LIN {X -0.115,Y -453.231,Z 768.523,A 0.000,B 0.000,C 90.000,E1 94.188} C_DIS
LIN {X 0.209,Y -441.249,Z 768.512,A 0.000,B 0.000,C 90.000,E1 92.064} C_DIS
LIN {X -0.076,Y -432.103,Z 768.503,A 0.000,B 0.000,C 90.000,E1 90.516} C_DIS
LIN {X -0.093,Y -422.619,Z 768.494,A 0.000,B 0.000,C 90.000,E1 88.912} C_DIS
LIN {X -0.178,Y -411.419,Z 768.483,A 0.000,B 0.000,C 90.000,E1 87.020} C_DIS
LIN {X -0.031,Y -400.090,Z 768.473,A 0.000,B 0.000,C 90.000,E1 85.065} C_DIS
LIN {X -0.072,Y -387.195,Z 768.460,A 0.000,B 0.000,C 90.000,E1 82.818} C_DIS
LIN {X 0.067,Y -373.104,Z 768.446,A 0.000,B 0.000,C 90.000,E1 80.208} C_DIS
LIN {X -0.105,Y -356.698,Z 768.428,A 0.000,B 0.000,C 90.000,E1 76.992} C_DIS
LIN {X -0.066,Y -345.249,Z 768.414,A 0.000,B 0.000,C 90.000,E1 74.574} C_DIS
LIN {X -0.147,Y -332.594,Z 768.399,A 0.000,B 0.000,C 90.000,E1 71.819} C_DIS
LIN {X 0.059,Y -320.333,Z 768.383,A 0.000,B 0.000,C 90.000,E1 68.954} C_DIS
LIN {X 0.088,Y -306.265,Z 768.363,A 0.000,B 0.000,C 90.000,E1 65.409} C_DIS
LIN {X 0.158,Y -293.532,Z 768.343,A 0.000,B 0.000,C 90.000,E1 61.769} C_DIS
LIN {X -0.092,Y -282.992,Z 768.325,A 0.000,B 0.000,C 90.000,E1 58.456} C_DIS
LIN {X 0.131,Y -275.046,Z 768.309,A 0.000,B 0.000,C 90.000,E1 55.674} C_DIS
LIN {X 0.000,Y -269.175,Z 768.298,A 0.000,B 0.000,C 90.000,E1 53.623} C_DIS
LIN {X 0.052,Y -261.369,Z 768.282,A 0.000,B 0.000,C 90.000,E1 50.803} C_DIS
LIN {X -0.041,Y -255.557,Z 768.270,A 0.000,B 0.000,C 90.000,E1 48.690} C_DIS
LIN {X -0.056,Y -247.855,Z 768.254,A 0.000,B 0.000,C 90.000,E1 45.810} C_DIS
LIN {X 0.075,Y -240.330,Z 768.238,A 0.000,B 0.000,C 90.000,E1 42.852} C_DIS
LIN {X 0.127,Y -231.043,Z 768.217,A 0.000,B 0.000,C 90.000,E1 39.116} C_DIS
LIN {X -0.014,Y -222.274,Z 768.196,A 0.000,B 0.000,C 90.000,E1 35.358} C_DIS
LIN {X 0.103,Y -214.211,Z 768.175,A 0.000,B 0.000,C 90.000,E1 31.465} C_DIS
LIN {X -0.013,Y -208.482,Z 768.158,A 0.000,B 0.000,C 90.000,E1 28.359} C_DIS
LIN {X 0.089,Y -203.532,Z 768.140,A 0.000,B 0.000,C 90.000,E1 25.155} C_DIS
LIN {X 0.040,Y -198.253,Z 768.118,A 0.000,B 0.000,C 90.000,E1 21.153} C_DIS
LIN {X 0.031,Y -194.129,Z 768.095,A 0.000,B 0.000,C 90.000,E1 17.094} C_DIS
LIN {X -0.008,Y -190.564,Z 768.068,A 0.000,B 0.000,C 90.000,E1 12.187} C_DIS
LIN {X 0.018,Y -188.134,Z 768.031,A 0.000,B 0.000,C 90.000,E1 5.568} C_DIS
LIN {X 0.043,Y -189.539,Z 767.970,A 0.000,B 0.000,C 90.000,E1 354.546} C_DIS
LIN {X -0.098,Y -193.008,Z 767.938,A 0.000,B 0.000,C 90.000,E1 348.814} C_DIS
LIN {X -0.033,Y -196.683,Z 767.915,A 0.000,B 0.000,C 90.000,E1 344.700} C_DIS
LIN {X 0.094,Y -201.414,Z 767.892,A 0.000,B 0.000,C 90.000,E1 340.604} C_DIS
LIN {X 0.009,Y -207.080,Z 767.870,A 0.000,B 0.000,C 90.000,E1 336.613} C_DIS
LIN {X -0.054,Y -213.642,Z 767.848,A 0.000,B 0.000,C 90.000,E1 332.666} C_DIS
LIN {X 0.008,Y -221.031,Z 767.826,A 0.000,B 0.000,C 90.000,E1 328.742} C_DIS
LIN {X 0.008,Y -228.997,Z 767.805,A 0.000,B 0.000,C 90.000,E1 324.895} C_DIS
LIN {X 0.108,Y -237.690,Z 767.784,A 0.000,B 0.000,C 90.000,E1 321.090} C_DIS
LIN {X 0.044,Y -247.109,Z 767.763,A 0.000,B 0.000,C 90.000,E1 317.391} C_DIS
LIN {X -0.092,Y -257.488,Z 767.743,A 0.000,B 0.000,C 90.000,E1 313.785} C_DIS
LIN {X 0.081,Y -267.584,Z 767.725,A 0.000,B 0.000,C 90.000,E1 310.539} C_DIS
LIN {X -0.049,Y -279.903,Z 767.706,A 0.000,B 0.000,C 90.000,E1 307.076} C_DIS
LIN {X 0.000,Y -293.440,Z 767.687,A 0.000,B 0.000,C 90.000,E1 303.658} C_DIS
LIN {X -0.087,Y -302.469,Z 767.676,A 0.000,B 0.000,C 90.000,E1 301.671} C_DIS
LIN {X 0.173,Y -319.454,Z 767.658,A 0.000,B 0.000,C 90.000,E1 298.359} C_DIS
LIN {X 0.007,Y -334.044,Z 767.644,A 0.000,B 0.000,C 90.000,E1 295.848} C_DIS
LIN {X 0.203,Y -345.763,Z 767.633,A 0.000,B 0.000,C 90.000,E1 293.951} C_DIS
LIN {X -0.078,Y -366.819,Z 767.616,A 0.000,B 0.000,C 90.000,E1 290.972} C_DIS
LIN {X -0.107,Y -390.144,Z 767.600,A 0.000,B 0.000,C 90.000,E1 288.055} C_DIS
LIN {X -0.085,Y -407.451,Z 767.589,A 0.000,B 0.000,C 90.000,E1 286.079} C_DIS
LIN {X 0.167,Y -419.629,Z 767.582,A 0.000,B 0.000,C 90.000,E1 284.662} C_DIS
LIN {X 0.199,Y -431.468,Z 767.574,A 0.000,B 0.000,C 90.000,E1 283.300} C_DIS
LIN {X -0.116,Y -442.966,Z 767.567,A 0.000,B 0.000,C 90.000,E1 282.007} C_DIS
LIN {X -0.085,Y -451.698,Z 767.561,A 0.000,B 0.000,C 90.000,E1 280.950} C_DIS
LIN {X 0.236,Y -461.835,Z 767.554,A 0.000,B 0.000,C 90.000,E1 279.613} C_DIS
LIN {X -0.050,Y -469.557,Z 767.548,A 0.000,B 0.000,C 90.000,E1 278.624} C_DIS
LIN {X -0.112,Y -475.010,Z 767.544,A 0.000,B 0.000,C 90.000,E1 277.871} C_DIS
LIN {X -0.194,Y -479.966,Z 767.539,A 0.000,B 0.000,C 90.000,E1 277.125} C_DIS
LIN {X -0.166,Y -484.180,Z 767.535,A 0.000,B 0.000,C 90.000,E1 276.372} C_DIS
LIN {X 0.012,Y -486.561,Z 767.533,A 0.000,B 0.000,C 90.000,E1 275.853} C_DIS
LIN {X 0.043,Y -489.431,Z 767.528,A 0.000,B 0.000,C 90.000,E1 275.106} C_DIS
LIN {X 0.251,Y -490.885,Z 767.526,A 0.000,B 0.000,C 90.000,E1 274.588} C_DIS
LIN {X -0.058,Y -491.996,Z 767.523,A 0.000,B 0.000,C 90.000,E1 274.131} C_DIS
LIN {X 0.168,Y -492.709,Z 767.520,A 0.000,B 0.000,C 90.000,E1 273.612} C_DIS
LIN {X -0.122,Y -493.040,Z 767.517,A 0.000,B 0.000,C 90.000,E1 273.154} C_DIS
LIN {X 0.111,Y -492.940,Z 767.515,A 0.000,B 0.000,C 90.000,E1 272.636} C_DIS
LIN {X -0.171,Y -492.377,Z 767.512,A 0.000,B 0.000,C 90.000,E1 272.178} C_DIS
LIN {X 0.057,Y -491.366,Z 767.509,A 0.000,B 0.000,C 90.000,E1 271.661} C_DIS
LIN {X -0.226,Y -489.879,Z 767.507,A 0.000,B 0.000,C 90.000,E1 271.203} C_DIS
LIN {X -0.023,Y -487.905,Z 767.504,A 0.000,B 0.000,C 90.000,E1 270.688} C_DIS
LIN {X 0.170,Y -485.305,Z 767.501,A 0.000,B 0.000,C 90.000,E1 270.172} C_DIS
LIN {X -0.139,Y -482.169,Z 767.498,A 0.000,B 0.000,C 90.000,E1 269.714} C_DIS
LIN {X 0.018,Y -478.202,Z 767.496,A 0.000,B 0.000,C 90.000,E1 269.198} C_DIS
LIN {X 0.152,Y -473.377,Z 767.493,A 0.000,B 0.000,C 90.000,E1 268.682} C_DIS
LIN {X -0.152,Y -467.577,Z 767.490,A 0.000,B 0.000,C 90.000,E1 268.224} C_DIS
LIN {X 0.054,Y -461.202,Z 767.488,A 0.000,B 0.000,C 90.000,E1 267.764} C_DIS
LIN {X -0.042,Y -457.997,Z 767.487,A 0.000,B 0.000,C 90.000,E1 267.593} C_DIS
LIN {X -0.137,Y -454.304,Z 767.486,A 0.000,B 0.000,C 90.000,E1 267.421} C_DIS
LIN {X -0.211,Y -446.988,Z 767.484,A 0.000,B 0.000,C 90.000,E1 267.135} C_DIS
LIN {X 0.167,Y -438.672,Z 767.483,A 0.000,B 0.000,C 90.000,E1 266.849} C_DIS
LIN {X -0.167,Y -429.640,Z 767.482,A 0.000,B 0.000,C 90.000,E1 266.731} C_DIS
LIN {X 0.129,Y -422.215,Z 767.481,A 0.000,B 0.000,C 90.000,E1 266.617} C_DIS
LIN {X 0.019,Y -417.823,Z 767.481,A 0.000,B 0.000,C 90.000,E1 266.617} C_DIS
LIN {X -0.015,Y -180.956,Z 767.481,A 0.000,B 0.000,C 90.000,E1 266.617} C_DIS
LIN {X 0.065,Y -180.879,Z 767.473,A 0.000,B 0.000,C 90.000,E1 265.065} C_DIS
LIN {X 0.006,Y -178.802,Z 767.442,A 0.000,B 0.000,C 90.000,E1 259.511} C_DIS
LIN {X 0.082,Y -175.847,Z 767.413,A 0.000,B 0.000,C 90.000,E1 254.393} C_DIS
LIN {X 0.042,Y -172.583,Z 767.390,A 0.000,B 0.000,C 90.000,E1 250.134} C_DIS
LIN {X 0.058,Y -171.470,Z 767.380,A 0.000,B 0.000,C 90.000,E1 248.411} C_DIS
LIN {X 0.038,Y -167.702,Z 767.356,A 0.000,B 0.000,C 90.000,E1 244.101} C_DIS
LIN {X 0.051,Y -166.387,Z 767.347,A 0.000,B 0.000,C 90.000,E1 242.359} C_DIS
LIN {X 0.042,Y -163.114,Z 767.327,A 0.000,B 0.000,C 90.000,E1 238.869} C_DIS
LIN {X 0.093,Y -161.064,Z 767.313,A 0.000,B 0.000,C 90.000,E1 236.215} C_DIS
LIN {X -0.021,Y -157.798,Z 767.293,A 0.000,B 0.000,C 90.000,E1 232.718} C_DIS
LIN {X 0.019,Y -155.834,Z 767.278,A 0.000,B 0.000,C 90.000,E1 230.033} C_DIS
LIN {X -0.024,Y -152.084,Z 767.253,A 0.000,B 0.000,C 90.000,E1 225.567} C_DIS
LIN {X -0.006,Y -150.334,Z 767.238,A 0.000,B 0.000,C 90.000,E1 222.852} C_DIS
LIN {X 0.015,Y -147.074,Z 767.213,A 0.000,B 0.000,C 90.000,E1 218.302} C_DIS
LIN {X -0.081,Y -145.648,Z 767.198,A 0.000,B 0.000,C 90.000,E1 215.598} C_DIS
LIN {X -0.077,Y -143.031,Z 767.172,A 0.000,B 0.000,C 90.000,E1 211.003} C_DIS
LIN {X 0.050,Y -141.656,Z 767.152,A 0.000,B 0.000,C 90.000,E1 207.257} C_DIS
LIN {X -0.031,Y -139.445,Z 767.115,A 0.000,B 0.000,C 90.000,E1 200.791} C_DIS
LIN {X 0.022,Y -139.179,Z 767.105,A 0.000,B 0.000,C 90.000,E1 198.906} C_DIS
LIN {X 0.050,Y -138.320,Z 767.053,A 0.000,B 0.000,C 90.000,E1 189.557} C_DIS
LIN {X 0.059,Y -139.466,Z 767.007,A 0.000,B 0.000,C 90.000,E1 181.146} C_DIS
LIN {X 0.001,Y -141.031,Z 766.975,A 0.000,B 0.000,C 90.000,E1 175.584} C_DIS
LIN {X -0.046,Y -142.398,Z 766.960,A 0.000,B 0.000,C 90.000,E1 172.818} C_DIS
LIN {X 0.017,Y -144.630,Z 766.934,A 0.000,B 0.000,C 90.000,E1 168.173} C_DIS
LIN {X 0.077,Y -147.825,Z 766.909,A 0.000,B 0.000,C 90.000,E1 163.559} C_DIS
LIN {X 0.022,Y -150.517,Z 766.889,A 0.000,B 0.000,C 90.000,E1 159.934} C_DIS
LIN {X 0.043,Y -153.979,Z 766.868,A 0.000,B 0.000,C 90.000,E1 156.305} C_DIS
LIN {X -0.037,Y -157.391,Z 766.849,A 0.000,B 0.000,C 90.000,E1 152.743} C_DIS
LIN {X 0.043,Y -161.596,Z 766.829,A 0.000,B 0.000,C 90.000,E1 149.154} C_DIS
LIN {X -0.085,Y -165.793,Z 766.809,A 0.000,B 0.000,C 90.000,E1 145.674} C_DIS
LIN {X 0.035,Y -170.756,Z 766.790,A 0.000,B 0.000,C 90.000,E1 142.145} C_DIS
LIN {X 0.058,Y -175.628,Z 766.771,A 0.000,B 0.000,C 90.000,E1 138.690} C_DIS
LIN {X -0.073,Y -181.243,Z 766.752,A 0.000,B 0.000,C 90.000,E1 135.324} C_DIS
LIN {X 0.058,Y -186.714,Z 766.733,A 0.000,B 0.000,C 90.000,E1 131.919} C_DIS
LIN {X 0.072,Y -191.544,Z 766.718,A 0.000,B 0.000,C 90.000,E1 129.277} C_DIS
LIN {X 0.081,Y -192.281,Z 766.716,A 0.000,B 0.000,C 90.000,E1 128.830} C_DIS
LIN {X 0.083,Y -291.983,Z 766.716,A 0.000,B 0.000,C 90.000,E1 128.830} C_DIS
LIN {X -0.037,Y -293.381,Z 766.716,A 0.000,B 0.000,C 90.000,E1 128.830} C_DIS
LIN {X -0.045,Y -297.878,Z 766.715,A 0.000,B 0.000,C 90.000,E1 128.624} C_DIS
LIN {X -0.048,Y -301.099,Z 766.713,A 0.000,B 0.000,C 90.000,E1 128.338} C_DIS
LIN {X 0.011,Y -304.766,Z 766.710,A 0.000,B 0.000,C 90.000,E1 127.810} C_DIS
LIN {X -0.036,Y -306.408,Z 766.708,A 0.000,B 0.000,C 90.000,E1 127.488} C_DIS
LIN {X -0.027,Y -307.697,Z 766.706,A 0.000,B 0.000,C 90.000,E1 127.156} C_DIS
LIN {X 0.075,Y -319.692,Z 766.685,A 0.000,B 0.000,C 90.000,E1 123.245} C_DIS
LIN {X 0.074,Y -330.066,Z 766.669,A 0.000,B 0.000,C 90.000,E1 120.384} C_DIS
LIN {X -0.017,Y -341.793,Z 766.653,A 0.000,B 0.000,C 90.000,E1 117.590} C_DIS
LIN {X 0.075,Y -354.971,Z 766.638,A 0.000,B 0.000,C 90.000,E1 114.823} C_DIS
LIN {X -0.138,Y -368.003,Z 766.625,A 0.000,B 0.000,C 90.000,E1 112.461} C_DIS
LIN {X -0.165,Y -382.370,Z 766.612,A 0.000,B 0.000,C 90.000,E1 110.120} C_DIS
LIN {X -0.096,Y -398.176,Z 766.599,A 0.000,B 0.000,C 90.000,E1 107.819} C_DIS
LIN {X 0.141,Y -415.535,Z 766.586,A 0.000,B 0.000,C 90.000,E1 105.552} C_DIS
LIN {X -0.101,Y -434.557,Z 766.574,A 0.000,B 0.000,C 90.000,E1 103.411} C_DIS
LIN {X -0.078,Y -454.655,Z 766.563,A 0.000,B 0.000,C 90.000,E1 101.366} C_DIS
LIN {X 0.205,Y -467.509,Z 766.556,A 0.000,B 0.000,C 90.000,E1 100.141} C_DIS
LIN {X -0.231,Y -469.681,Z 766.555,A 0.000,B 0.000,C 90.000,E1 99.962} C_DIS
LIN {X -0.207,Y -471.323,Z 766.554,A 0.000,B 0.000,C 90.000,E1 99.726} C_DIS
LIN {X 0.033,Y -472.685,Z 766.552,A 0.000,B 0.000,C 90.000,E1 99.443} C_DIS
LIN {X -0.113,Y -473.694,Z 766.551,A 0.000,B 0.000,C 90.000,E1 99.208} C_DIS
LIN {X 0.074,Y -474.848,Z 766.548,A 0.000,B 0.000,C 90.000,E1 98.681} C_DIS
LIN {X 0.194,Y -475.004,Z 766.545,A 0.000,B 0.000,C 90.000,E1 98.163} C_DIS
LIN {X -0.147,Y -474.191,Z 766.543,A 0.000,B 0.000,C 90.000,E1 97.701} C_DIS
LIN {X -0.015,Y -472.276,Z 766.540,A 0.000,B 0.000,C 90.000,E1 97.182} C_DIS
LIN {X 0.113,Y -469.117,Z 766.537,A 0.000,B 0.000,C 90.000,E1 96.663} C_DIS
LIN {X 0.197,Y -451.453,Z 766.521,A 0.000,B 0.000,C 90.000,E1 93.841} C_DIS
LIN {X -0.173,Y -441.001,Z 766.511,A 0.000,B 0.000,C 90.000,E1 92.064} C_DIS
LIN {X -0.022,Y -431.870,Z 766.503,A 0.000,B 0.000,C 90.000,E1 90.458} C_DIS
LIN {X -0.044,Y -422.368,Z 766.494,A 0.000,B 0.000,C 90.000,E1 88.854} C_DIS
LIN {X -0.137,Y -411.187,Z 766.483,A 0.000,B 0.000,C 90.000,E1 86.963} C_DIS
LIN {X 0.004,Y -399.867,Z 766.472,A 0.000,B 0.000,C 90.000,E1 85.008} C_DIS
LIN {X -0.045,Y -386.980,Z 766.460,A 0.000,B 0.000,C 90.000,E1 82.761} C_DIS
LIN {X 0.092,Y -371.356,Z 766.444,A 0.000,B 0.000,C 90.000,E1 79.859} C_DIS
LIN {X -0.098,Y -356.521,Z 766.427,A 0.000,B 0.000,C 90.000,E1 76.937} C_DIS
LIN {X -0.067,Y -345.091,Z 766.414,A 0.000,B 0.000,C 90.000,E1 74.519} C_DIS
LIN {X -0.157,Y -332.443,Z 766.399,A 0.000,B 0.000,C 90.000,E1 71.764} C_DIS
LIN {X 0.040,Y -320.223,Z 766.383,A 0.000,B 0.000,C 90.000,E1 68.901} C_DIS
LIN {X 0.059,Y -306.215,Z 766.363,A 0.000,B 0.000,C 90.000,E1 65.357} C_DIS
LIN {X -0.137,Y -293.572,Z 766.343,A 0.000,B 0.000,C 90.000,E1 61.769} C_DIS
LIN {X -0.134,Y -283.092,Z 766.324,A 0.000,B 0.000,C 90.000,E1 58.408} C_DIS
LIN {X -0.140,Y -275.193,Z 766.309,A 0.000,B 0.000,C 90.000,E1 55.674} C_DIS
LIN {X 0.118,Y -267.422,Z 766.294,A 0.000,B 0.000,C 90.000,E1 52.844} C_DIS
LIN {X 0.169,Y -261.602,Z 766.282,A 0.000,B 0.000,C 90.000,E1 50.723} C_DIS
LIN {X 0.077,Y -255.815,Z 766.270,A 0.000,B 0.000,C 90.000,E1 48.609} C_DIS
LIN {X 0.066,Y -248.116,Z 766.254,A 0.000,B 0.000,C 90.000,E1 45.729} C_DIS
LIN {X 0.025,Y -240.586,Z 766.238,A 0.000,B 0.000,C 90.000,E1 42.813} C_DIS
LIN {X -0.006,Y -233.076,Z 766.221,A 0.000,B 0.000,C 90.000,E1 39.850} C_DIS
LIN {X 0.031,Y -225.925,Z 766.205,A 0.000,B 0.000,C 90.000,E1 36.824} C_DIS
LIN {X -0.032,Y -217.524,Z 766.183,A 0.000,B 0.000,C 90.000,E1 33.007} C_DIS
LIN {X 0.039,Y -211.441,Z 766.166,A 0.000,B 0.000,C 90.000,E1 29.873} C_DIS
LIN {X -0.058,Y -206.090,Z 766.148,A 0.000,B 0.000,C 90.000,E1 26.744} C_DIS
LIN {X 0.060,Y -200.405,Z 766.126,A 0.000,B 0.000,C 90.000,E1 22.717} C_DIS
LIN {X 0.072,Y -195.833,Z 766.104,A 0.000,B 0.000,C 90.000,E1 18.671} C_DIS
LIN {X 0.060,Y -192.317,Z 766.081,A 0.000,B 0.000,C 90.000,E1 14.592} C_DIS
LIN {X -0.041,Y -189.168,Z 766.049,A 0.000,B 0.000,C 90.000,E1 8.859} C_DIS
LIN {X -0.028,Y -190.058,Z 765.965,A 0.000,B 0.000,C 90.000,E1 353.742} C_DIS
LIN {X -0.087,Y -193.131,Z 765.938,A 0.000,B 0.000,C 90.000,E1 348.814} C_DIS
LIN {X -0.018,Y -196.809,Z 765.915,A 0.000,B 0.000,C 90.000,E1 344.700} C_DIS
LIN {X 0.113,Y -201.538,Z 765.892,A 0.000,B 0.000,C 90.000,E1 340.604} C_DIS
LIN {X 0.032,Y -207.205,Z 765.870,A 0.000,B 0.000,C 90.000,E1 336.613} C_DIS
LIN {X -0.027,Y -213.763,Z 765.848,A 0.000,B 0.000,C 90.000,E1 332.666} C_DIS
LIN {X 0.040,Y -221.120,Z 765.826,A 0.000,B 0.000,C 90.000,E1 328.742} C_DIS
LIN {X 0.045,Y -229.078,Z 765.805,A 0.000,B 0.000,C 90.000,E1 324.895} C_DIS
LIN {X -0.001,Y -237.750,Z 765.784,A 0.000,B 0.000,C 90.000,E1 321.126} C_DIS
LIN {X 0.089,Y -247.144,Z 765.763,A 0.000,B 0.000,C 90.000,E1 317.391} C_DIS
LIN {X -0.044,Y -257.529,Z 765.743,A 0.000,B 0.000,C 90.000,E1 313.785} C_DIS
LIN {X 0.131,Y -267.596,Z 765.725,A 0.000,B 0.000,C 90.000,E1 310.539} C_DIS
LIN {X 0.004,Y -279.903,Z 765.706,A 0.000,B 0.000,C 90.000,E1 307.076} C_DIS
LIN {X 0.056,Y -293.422,Z 765.687,A 0.000,B 0.000,C 90.000,E1 303.658} C_DIS
LIN {X -0.031,Y -302.437,Z 765.676,A 0.000,B 0.000,C 90.000,E1 301.671} C_DIS
LIN {X -0.050,Y -319.412,Z 765.658,A 0.000,B 0.000,C 90.000,E1 298.409} C_DIS
LIN {X 0.032,Y -335.868,Z 765.642,A 0.000,B 0.000,C 90.000,E1 295.540} C_DIS
LIN {X 0.045,Y -355.974,Z 765.625,A 0.000,B 0.000,C 90.000,E1 292.461} C_DIS
LIN {X -0.157,Y -375.747,Z 765.610,A 0.000,B 0.000,C 90.000,E1 289.812} C_DIS
LIN {X 0.051,Y -399.750,Z 765.594,A 0.000,B 0.000,C 90.000,E1 286.913} C_DIS
LIN {X -0.113,Y -412.105,Z 765.586,A 0.000,B 0.000,C 90.000,E1 285.536} C_DIS
LIN {X 0.208,Y -424.131,Z 765.579,A 0.000,B 0.000,C 90.000,E1 284.120} C_DIS
LIN {X -0.221,Y -435.815,Z 765.571,A 0.000,B 0.000,C 90.000,E1 282.827} C_DIS
LIN {X 0.160,Y -444.933,Z 765.565,A 0.000,B 0.000,C 90.000,E1 281.715} C_DIS
LIN {X 0.219,Y -453.492,Z 765.559,A 0.000,B 0.000,C 90.000,E1 280.658} C_DIS
LIN {X 0.124,Y -463.520,Z 765.552,A 0.000,B 0.000,C 90.000,E1 279.378} C_DIS
LIN {X -0.219,Y -471.181,Z 765.547,A 0.000,B 0.000,C 90.000,E1 278.398} C_DIS
LIN {X 0.202,Y -476.526,Z 765.542,A 0.000,B 0.000,C 90.000,E1 277.587} C_DIS
LIN {X 0.204,Y -481.299,Z 765.538,A 0.000,B 0.000,C 90.000,E1 276.834} C_DIS
LIN {X 0.186,Y -485.273,Z 765.534,A 0.000,B 0.000,C 90.000,E1 276.087} C_DIS
LIN {X -0.108,Y -487.531,Z 765.531,A 0.000,B 0.000,C 90.000,E1 275.625} C_DIS
LIN {X 0.094,Y -489.377,Z 765.528,A 0.000,B 0.000,C 90.000,E1 275.106} C_DIS
LIN {X -0.187,Y -490.862,Z 765.526,A 0.000,B 0.000,C 90.000,E1 274.645} C_DIS
LIN {X -0.006,Y -492.002,Z 765.523,A 0.000,B 0.000,C 90.000,E1 274.131} C_DIS
LIN {X 0.219,Y -492.762,Z 765.520,A 0.000,B 0.000,C 90.000,E1 273.612} C_DIS
LIN {X -0.071,Y -493.127,Z 765.517,A 0.000,B 0.000,C 90.000,E1 273.154} C_DIS
LIN {X 0.162,Y -493.046,Z 765.515,A 0.000,B 0.000,C 90.000,E1 272.636} C_DIS
LIN {X -0.119,Y -492.562,Z 765.512,A 0.000,B 0.000,C 90.000,E1 272.178} C_DIS
LIN {X 0.109,Y -491.565,Z 765.509,A 0.000,B 0.000,C 90.000,E1 271.661} C_DIS
LIN {X -0.173,Y -490.119,Z 765.507,A 0.000,B 0.000,C 90.000,E1 271.203} C_DIS
LIN {X 0.031,Y -488.140,Z 765.504,A 0.000,B 0.000,C 90.000,E1 270.688} C_DIS
LIN {X 0.225,Y -485.587,Z 765.501,A 0.000,B 0.000,C 90.000,E1 270.172} C_DIS
LIN {X -0.083,Y -482.401,Z 765.498,A 0.000,B 0.000,C 90.000,E1 269.714} C_DIS
LIN {X 0.076,Y -478.460,Z 765.496,A 0.000,B 0.000,C 90.000,E1 269.198} C_DIS
LIN {X 0.211,Y -473.627,Z 765.493,A 0.000,B 0.000,C 90.000,E1 268.682} C_DIS
LIN {X 0.081,Y -470.963,Z 765.491,A 0.000,B 0.000,C 90.000,E1 268.453} C_DIS
LIN {X 0.062,Y -465.020,Z 765.489,A 0.000,B 0.000,C 90.000,E1 267.993} C_DIS
LIN {X 0.046,Y -458.501,Z 765.487,A 0.000,B 0.000,C 90.000,E1 267.593} C_DIS
LIN {X 0.125,Y -451.362,Z 765.485,A 0.000,B 0.000,C 90.000,E1 267.249} C_DIS
LIN {X -0.140,Y -447.619,Z 765.484,A 0.000,B 0.000,C 90.000,E1 267.135} C_DIS
LIN {X 0.199,Y -439.329,Z 765.483,A 0.000,B 0.000,C 90.000,E1 266.849} C_DIS
LIN {X -0.167,Y -430.566,Z 765.482,A 0.000,B 0.000,C 90.000,E1 266.731} C_DIS
LIN {X 0.112,Y -423.768,Z 765.481,A 0.000,B 0.000,C 90.000,E1 266.617} C_DIS
LIN {X -0.065,Y -419.400,Z 765.481,A 0.000,B 0.000,C 90.000,E1 266.617} C_DIS
LIN {X -0.053,Y -180.956,Z 765.481,A 0.000,B 0.000,C 90.000,E1 266.617} C_DIS
LIN {X 0.026,Y -180.877,Z 765.473,A 0.000,B 0.000,C 90.000,E1 265.065} C_DIS
LIN {X -0.032,Y -178.795,Z 765.442,A 0.000,B 0.000,C 90.000,E1 259.511} C_DIS
LIN {X 0.044,Y -175.840,Z 765.413,A 0.000,B 0.000,C 90.000,E1 254.393} C_DIS
LIN {X 0.044,Y -172.032,Z 765.385,A 0.000,B 0.000,C 90.000,E1 249.263} C_DIS
LIN {X 0.020,Y -171.460,Z 765.380,A 0.000,B 0.000,C 90.000,E1 248.411} C_DIS
LIN {X 0.000,Y -167.692,Z 765.356,A 0.000,B 0.000,C 90.000,E1 244.101} C_DIS
LIN {X 0.014,Y -166.375,Z 765.346,A 0.000,B 0.000,C 90.000,E1 242.359} C_DIS
LIN {X 0.005,Y -163.104,Z 765.327,A 0.000,B 0.000,C 90.000,E1 238.869} C_DIS
LIN {X 0.056,Y -161.051,Z 765.312,A 0.000,B 0.000,C 90.000,E1 236.215} C_DIS
LIN {X 0.039,Y -157.787,Z 765.293,A 0.000,B 0.000,C 90.000,E1 232.683} C_DIS
LIN {X -0.017,Y -155.823,Z 765.278,A 0.000,B 0.000,C 90.000,E1 230.033} C_DIS
LIN {X -0.060,Y -152.074,Z 765.253,A 0.000,B 0.000,C 90.000,E1 225.567} C_DIS
LIN {X -0.041,Y -150.325,Z 765.238,A 0.000,B 0.000,C 90.000,E1 222.852} C_DIS
LIN {X -0.020,Y -147.066,Z 765.213,A 0.000,B 0.000,C 90.000,E1 218.302} C_DIS
LIN {X 0.088,Y -145.642,Z 765.198,A 0.000,B 0.000,C 90.000,E1 215.518} C_DIS
LIN {X 0.086,Y -143.025,Z 765.172,A 0.000,B 0.000,C 90.000,E1 210.924} C_DIS
LIN {X 0.017,Y -141.650,Z 765.151,A 0.000,B 0.000,C 90.000,E1 207.257} C_DIS
LIN {X -0.063,Y -139.444,Z 765.115,A 0.000,B 0.000,C 90.000,E1 200.791} C_DIS
LIN {X -0.011,Y -139.177,Z 765.105,A 0.000,B 0.000,C 90.000,E1 198.906} C_DIS
LIN {X 0.017,Y -138.319,Z 765.053,A 0.000,B 0.000,C 90.000,E1 189.557} C_DIS
LIN {X 0.026,Y -139.468,Z 765.006,A 0.000,B 0.000,C 90.000,E1 181.146} C_DIS
LIN {X -0.033,Y -141.036,Z 764.975,A 0.000,B 0.000,C 90.000,E1 175.584} C_DIS
LIN {X 0.062,Y -142.404,Z 764.960,A 0.000,B 0.000,C 90.000,E1 172.761} C_DIS
LIN {X -0.017,Y -144.638,Z 764.934,A 0.000,B 0.000,C 90.000,E1 168.173} C_DIS
LIN {X 0.043,Y -147.834,Z 764.909,A 0.000,B 0.000,C 90.000,E1 163.559} C_DIS
LIN {X -0.013,Y -150.529,Z 764.888,A 0.000,B 0.000,C 90.000,E1 159.934} C_DIS
LIN {X 0.007,Y -153.992,Z 764.868,A 0.000,B 0.000,C 90.000,E1 156.305} C_DIS
LIN {X -0.073,Y -157.406,Z 764.848,A 0.000,B 0.000,C 90.000,E1 152.743} C_DIS
LIN {X 0.007,Y -161.613,Z 764.829,A 0.000,B 0.000,C 90.000,E1 149.154} C_DIS
LIN {X 0.108,Y -165.809,Z 764.809,A 0.000,B 0.000,C 90.000,E1 145.595} C_DIS
LIN {X -0.003,Y -170.775,Z 764.790,A 0.000,B 0.000,C 90.000,E1 142.145} C_DIS
LIN {X 0.020,Y -175.647,Z 764.771,A 0.000,B 0.000,C 90.000,E1 138.690} C_DIS
LIN {X 0.018,Y -181.261,Z 764.752,A 0.000,B 0.000,C 90.000,E1 135.283} C_DIS
LIN {X 0.017,Y -186.735,Z 764.733,A 0.000,B 0.000,C 90.000,E1 131.919} C_DIS
LIN {X 0.032,Y -191.563,Z 764.718,A 0.000,B 0.000,C 90.000,E1 129.277} C_DIS
LIN {X -0.105,Y -192.238,Z 764.716,A 0.000,B 0.000,C 90.000,E1 128.910} C_DIS
LIN {X -0.022,Y -291.703,Z 764.716,A 0.000,B 0.000,C 90.000,E1 128.874} C_DIS
LIN {X 0.068,Y -293.365,Z 764.716,A 0.000,B 0.000,C 90.000,E1 128.830} C_DIS
LIN {X -0.108,Y -298.260,Z 764.714,A 0.000,B 0.000,C 90.000,E1 128.624} C_DIS
LIN {X -0.013,Y -301.459,Z 764.713,A 0.000,B 0.000,C 90.000,E1 128.302} C_DIS
LIN {X 0.139,Y -305.106,Z 764.710,A 0.000,B 0.000,C 90.000,E1 127.729} C_DIS
LIN {X -0.094,Y -306.656,Z 764.708,A 0.000,B 0.000,C 90.000,E1 127.443} C_DIS
LIN {X 0.103,Y -307.876,Z 764.706,A 0.000,B 0.000,C 90.000,E1 127.076} C_DIS
LIN {X 0.141,Y -318.779,Z 764.686,A 0.000,B 0.000,C 90.000,E1 123.499} C_DIS
LIN {X -0.062,Y -329.035,Z 764.670,A 0.000,B 0.000,C 90.000,E1 120.669} C_DIS
LIN {X -0.015,Y -340.630,Z 764.655,A 0.000,B 0.000,C 90.000,E1 117.847} C_DIS
LIN {X 0.040,Y -353.673,Z 764.639,A 0.000,B 0.000,C 90.000,E1 115.079} C_DIS
LIN {X -0.062,Y -366.572,Z 764.626,A 0.000,B 0.000,C 90.000,E1 112.695} C_DIS
LIN {X -0.132,Y -380.797,Z 764.613,A 0.000,B 0.000,C 90.000,E1 110.355} C_DIS
LIN {X -0.107,Y -396.448,Z 764.600,A 0.000,B 0.000,C 90.000,E1 108.055} C_DIS
LIN {X 0.079,Y -413.641,Z 764.588,A 0.000,B 0.000,C 90.000,E1 105.788} C_DIS
LIN {X 0.196,Y -432.500,Z 764.576,A 0.000,B 0.000,C 90.000,E1 103.592} C_DIS
LIN {X 0.182,Y -452.537,Z 764.564,A 0.000,B 0.000,C 90.000,E1 101.535} C_DIS
LIN {X -0.123,Y -467.906,Z 764.556,A 0.000,B 0.000,C 90.000,E1 100.141} C_DIS
LIN {X -0.106,Y -469.984,Z 764.555,A 0.000,B 0.000,C 90.000,E1 99.905} C_DIS
LIN {X -0.089,Y -471.563,Z 764.554,A 0.000,B 0.000,C 90.000,E1 99.670} C_DIS
LIN {X 0.231,Y -472.864,Z 764.552,A 0.000,B 0.000,C 90.000,E1 99.378} C_DIS
LIN {X 0.008,Y -473.824,Z 764.551,A 0.000,B 0.000,C 90.000,E1 99.151} C_DIS
LIN {X 0.197,Y -474.897,Z 764.548,A 0.000,B 0.000,C 90.000,E1 98.624} C_DIS
LIN {X -0.151,Y -474.979,Z 764.545,A 0.000,B 0.000,C 90.000,E1 98.163} C_DIS
LIN {X -0.020,Y -474.089,Z 764.542,A 0.000,B 0.000,C 90.000,E1 97.644} C_DIS
LIN {X 0.111,Y -472.078,Z 764.540,A 0.000,B 0.000,C 90.000,E1 97.125} C_DIS
LIN {X 0.177,Y -463.915,Z 764.533,A 0.000,B 0.000,C 90.000,E1 95.853} C_DIS
LIN {X 0.074,Y -449.731,Z 764.520,A 0.000,B 0.000,C 90.000,E1 93.555} C_DIS
LIN {X -0.065,Y -440.789,Z 764.511,A 0.000,B 0.000,C 90.000,E1 92.007} C_DIS
LIN {X 0.081,Y -431.669,Z 764.502,A 0.000,B 0.000,C 90.000,E1 90.401} C_DIS
LIN {X 0.052,Y -422.159,Z 764.493,A 0.000,B 0.000,C 90.000,E1 88.797} C_DIS
LIN {X -0.047,Y -410.990,Z 764.483,A 0.000,B 0.000,C 90.000,E1 86.906} C_DIS
LIN {X 0.086,Y -399.688,Z 764.472,A 0.000,B 0.000,C 90.000,E1 84.951} C_DIS
LIN {X 0.029,Y -386.806,Z 764.459,A 0.000,B 0.000,C 90.000,E1 82.704} C_DIS
LIN {X 0.149,Y -372.755,Z 764.445,A 0.000,B 0.000,C 90.000,E1 80.095} C_DIS
LIN {X -0.045,Y -356.390,Z 764.427,A 0.000,B 0.000,C 90.000,E1 76.881} C_DIS
LIN {X 0.069,Y -344.968,Z 764.414,A 0.000,B 0.000,C 90.000,E1 74.448} C_DIS
LIN {X 0.000,Y -333.706,Z 764.400,A 0.000,B 0.000,C 90.000,E1 72.000} C_DIS
LIN {X -0.187,Y -321.457,Z 764.384,A 0.000,B 0.000,C 90.000,E1 69.209} C_DIS
LIN {X -0.111,Y -307.411,Z 764.365,A 0.000,B 0.000,C 90.000,E1 65.665} C_DIS
LIN {X 0.002,Y -294.718,Z 764.345,A 0.000,B 0.000,C 90.000,E1 62.025} C_DIS
LIN {X 0.059,Y -285.239,Z 764.328,A 0.000,B 0.000,C 90.000,E1 58.997} C_DIS
LIN {X -0.047,Y -277.332,Z 764.313,A 0.000,B 0.000,C 90.000,E1 56.294} C_DIS
LIN {X 0.107,Y -269.562,Z 764.297,A 0.000,B 0.000,C 90.000,E1 53.497} C_DIS
LIN {X 0.033,Y -263.787,Z 764.286,A 0.000,B 0.000,C 90.000,E1 51.412} C_DIS
LIN {X 0.068,Y -256.083,Z 764.270,A 0.000,B 0.000,C 90.000,E1 48.566} C_DIS
LIN {X -0.122,Y -248.398,Z 764.254,A 0.000,B 0.000,C 90.000,E1 45.729} C_DIS
LIN {X -0.126,Y -242.738,Z 764.242,A 0.000,B 0.000,C 90.000,E1 43.542} C_DIS
LIN {X 0.062,Y -235.183,Z 764.225,A 0.000,B 0.000,C 90.000,E1 40.539} C_DIS
LIN {X 0.012,Y -226.161,Z 764.204,A 0.000,B 0.000,C 90.000,E1 36.790} C_DIS
LIN {X 0.105,Y -219.351,Z 764.187,A 0.000,B 0.000,C 90.000,E1 33.706} C_DIS
LIN {X 0.039,Y -213.104,Z 764.170,A 0.000,B 0.000,C 90.000,E1 30.620} C_DIS
LIN {X -0.099,Y -207.549,Z 764.153,A 0.000,B 0.000,C 90.000,E1 27.513} C_DIS
LIN {X -0.037,Y -201.657,Z 764.131,A 0.000,B 0.000,C 90.000,E1 23.515} C_DIS
LIN {X 0.077,Y -196.834,Z 764.108,A 0.000,B 0.000,C 90.000,E1 19.450} C_DIS
LIN {X -0.091,Y -193.117,Z 764.086,A 0.000,B 0.000,C 90.000,E1 15.426} C_DIS
LIN {X -0.064,Y -190.013,Z 764.058,A 0.000,B 0.000,C 90.000,E1 10.489} C_DIS
LIN {X -0.027,Y -188.127,Z 764.008,A 0.000,B 0.000,C 90.000,E1 1.375} C_DIS
LIN {X -0.023,Y -190.184,Z 763.965,A 0.000,B 0.000,C 90.000,E1 353.742} C_DIS
LIN {X -0.077,Y -193.238,Z 763.938,A 0.000,B 0.000,C 90.000,E1 348.814} C_DIS
LIN {X -0.004,Y -196.930,Z 763.915,A 0.000,B 0.000,C 90.000,E1 344.700} C_DIS
LIN {X -0.060,Y -201.649,Z 763.892,A 0.000,B 0.000,C 90.000,E1 340.659} C_DIS
LIN {X 0.054,Y -207.334,Z 763.870,A 0.000,B 0.000,C 90.000,E1 336.613} C_DIS
LIN {X 0.000,Y -213.875,Z 763.848,A 0.000,B 0.000,C 90.000,E1 332.666} C_DIS
LIN {X 0.071,Y -221.203,Z 763.826,A 0.000,B 0.000,C 90.000,E1 328.742} C_DIS
LIN {X 0.020,Y -227.537,Z 763.809,A 0.000,B 0.000,C 90.000,E1 325.674} C_DIS
LIN {X -0.076,Y -235.996,Z 763.788,A 0.000,B 0.000,C 90.000,E1 321.904} C_DIS
LIN {X -0.015,Y -245.211,Z 763.768,A 0.000,B 0.000,C 90.000,E1 318.162} C_DIS
LIN {X -0.037,Y -255.416,Z 763.747,A 0.000,B 0.000,C 90.000,E1 314.514} C_DIS
LIN {X 0.114,Y -266.452,Z 763.727,A 0.000,B 0.000,C 90.000,E1 310.906} C_DIS
LIN {X -0.052,Y -278.615,Z 763.708,A 0.000,B 0.000,C 90.000,E1 307.443} C_DIS
LIN {X 0.120,Y -291.996,Z 763.689,A 0.000,B 0.000,C 90.000,E1 303.992} C_DIS
LIN {X 0.021,Y -302.427,Z 763.676,A 0.000,B 0.000,C 90.000,E1 301.671} C_DIS
LIN {X 0.004,Y -319.360,Z 763.658,A 0.000,B 0.000,C 90.000,E1 298.409} C_DIS
LIN {X 0.122,Y -333.950,Z 763.644,A 0.000,B 0.000,C 90.000,E1 295.848} C_DIS
LIN {X 0.008,Y -347.628,Z 763.632,A 0.000,B 0.000,C 90.000,E1 293.695} C_DIS
LIN {X 0.067,Y -371.081,Z 763.613,A 0.000,B 0.000,C 90.000,E1 290.375} C_DIS
LIN {X -0.142,Y -397.162,Z 763.596,A 0.000,B 0.000,C 90.000,E1 287.221} C_DIS
LIN {X 0.057,Y -409.539,Z 763.588,A 0.000,B 0.000,C 90.000,E1 285.788} C_DIS
LIN {X 0.039,Y -421.601,Z 763.580,A 0.000,B 0.000,C 90.000,E1 284.411} C_DIS
LIN {X -0.004,Y -433.324,Z 763.573,A 0.000,B 0.000,C 90.000,E1 283.063} C_DIS
LIN {X 0.129,Y -444.742,Z 763.565,A 0.000,B 0.000,C 90.000,E1 281.715} C_DIS
LIN {X 0.186,Y -453.270,Z 763.559,A 0.000,B 0.000,C 90.000,E1 280.658} C_DIS
LIN {X 0.086,Y -463.324,Z 763.552,A 0.000,B 0.000,C 90.000,E1 279.378} C_DIS
LIN {X 0.208,Y -471.017,Z 763.546,A 0.000,B 0.000,C 90.000,E1 278.341} C_DIS
LIN {X 0.020,Y -478.054,Z 763.541,A 0.000,B 0.000,C 90.000,E1 277.352} C_DIS
LIN {X 0.160,Y -481.178,Z 763.538,A 0.000,B 0.000,C 90.000,E1 276.834} C_DIS
LIN {X 0.141,Y -485.206,Z 763.534,A 0.000,B 0.000,C 90.000,E1 276.087} C_DIS
LIN {X -0.154,Y -487.483,Z 763.531,A 0.000,B 0.000,C 90.000,E1 275.625} C_DIS
LIN {X 0.048,Y -489.361,Z 763.528,A 0.000,B 0.000,C 90.000,E1 275.106} C_DIS
LIN {X -0.235,Y -490.902,Z 763.526,A 0.000,B 0.000,C 90.000,E1 274.645} C_DIS
LIN {X -0.054,Y -492.047,Z 763.523,A 0.000,B 0.000,C 90.000,E1 274.131} C_DIS
LIN {X 0.172,Y -492.820,Z 763.520,A 0.000,B 0.000,C 90.000,E1 273.612} C_DIS
LIN {X -0.118,Y -493.227,Z 763.517,A 0.000,B 0.000,C 90.000,E1 273.154} C_DIS
LIN {X 0.116,Y -493.170,Z 763.515,A 0.000,B 0.000,C 90.000,E1 272.636} C_DIS
LIN {X -0.164,Y -492.685,Z 763.512,A 0.000,B 0.000,C 90.000,E1 272.178} C_DIS
LIN {X 0.064,Y -491.734,Z 763.509,A 0.000,B 0.000,C 90.000,E1 271.661} C_DIS
LIN {X -0.218,Y -490.296,Z 763.507,A 0.000,B 0.000,C 90.000,E1 271.203} C_DIS
LIN {X -0.158,Y -487.154,Z 763.502,A 0.000,B 0.000,C 90.000,E1 270.458} C_DIS
LIN {X 0.029,Y -484.288,Z 763.500,A 0.000,B 0.000,C 90.000,E1 269.943} C_DIS
LIN {X 0.197,Y -480.726,Z 763.497,A 0.000,B 0.000,C 90.000,E1 269.427} C_DIS
LIN {X -0.132,Y -476.338,Z 763.494,A 0.000,B 0.000,C 90.000,E1 268.969} C_DIS
LIN {X 0.051,Y -471.153,Z 763.491,A 0.000,B 0.000,C 90.000,E1 268.453} C_DIS
LIN {X -0.072,Y -468.189,Z 763.490,A 0.000,B 0.000,C 90.000,E1 268.224} C_DIS
LIN {X 0.119,Y -461.900,Z 763.488,A 0.000,B 0.000,C 90.000,E1 267.764} C_DIS
LIN {X -0.121,Y -454.925,Z 763.486,A 0.000,B 0.000,C 90.000,E1 267.421} C_DIS
LIN {X -0.221,Y -447.671,Z 763.484,A 0.000,B 0.000,C 90.000,E1 267.135} C_DIS
LIN {X 0.132,Y -439.555,Z 763.483,A 0.000,B 0.000,C 90.000,E1 266.849} C_DIS
LIN {X 0.180,Y -430.567,Z 763.482,A 0.000,B 0.000,C 90.000,E1 266.674} C_DIS
LIN {X -0.005,Y -423.409,Z 763.481,A 0.000,B 0.000,C 90.000,E1 266.617} C_DIS
LIN {X 0.212,Y -417.182,Z 763.481,A 0.000,B 0.000,C 90.000,E1 266.560} C_DIS
LIN {X 0.071,Y -180.954,Z 763.481,A 0.000,B 0.000,C 90.000,E1 266.560} C_DIS
LIN {X 0.039,Y -180.821,Z 763.471,A 0.000,B 0.000,C 90.000,E1 264.837} C_DIS
LIN {X -0.061,Y -178.925,Z 763.443,A 0.000,B 0.000,C 90.000,E1 259.803} C_DIS
LIN {X -0.022,Y -175.971,Z 763.415,A 0.000,B 0.000,C 90.000,E1 254.700} C_DIS
LIN {X -0.028,Y -175.456,Z 763.410,A 0.000,B 0.000,C 90.000,E1 253.850} C_DIS
LIN {X -0.020,Y -172.208,Z 763.386,A 0.000,B 0.000,C 90.000,E1 249.571} C_DIS
LIN {X -0.041,Y -171.683,Z 763.382,A 0.000,B 0.000,C 90.000,E1 248.720} C_DIS
LIN {X -0.050,Y -167.909,Z 763.358,A 0.000,B 0.000,C 90.000,E1 244.409} C_DIS
LIN {X -0.032,Y -166.650,Z 763.348,A 0.000,B 0.000,C 90.000,E1 242.666} C_DIS
LIN {X 0.023,Y -162.634,Z 763.324,A 0.000,B 0.000,C 90.000,E1 238.280} C_DIS
LIN {X 0.082,Y -161.322,Z 763.314,A 0.000,B 0.000,C 90.000,E1 236.501} C_DIS
LIN {X -0.009,Y -157.318,Z 763.289,A 0.000,B 0.000,C 90.000,E1 232.110} C_DIS
LIN {X -0.077,Y -155.297,Z 763.275,A 0.000,B 0.000,C 90.000,E1 229.461} C_DIS
LIN {X 0.070,Y -151.657,Z 763.250,A 0.000,B 0.000,C 90.000,E1 224.919} C_DIS
LIN {X 0.007,Y -150.525,Z 763.240,A 0.000,B 0.000,C 90.000,E1 223.137} C_DIS
LIN {X 0.029,Y -147.249,Z 763.214,A 0.000,B 0.000,C 90.000,E1 218.588} C_DIS
LIN {X -0.006,Y -145.274,Z 763.194,A 0.000,B 0.000,C 90.000,E1 214.945} C_DIS
LIN {X 0.029,Y -142.380,Z 763.163,A 0.000,B 0.000,C 90.000,E1 209.411} C_DIS
LIN {X -0.049,Y -141.357,Z 763.148,A 0.000,B 0.000,C 90.000,E1 206.668} C_DIS
LIN {X 0.061,Y -139.341,Z 763.112,A 0.000,B 0.000,C 90.000,E1 200.120} C_DIS
LIN {X -0.021,Y -139.009,Z 763.102,A 0.000,B 0.000,C 90.000,E1 198.290} C_DIS
LIN {X -0.070,Y -138.340,Z 763.055,A 0.000,B 0.000,C 90.000,E1 189.905} C_DIS
LIN {X -0.050,Y -139.401,Z 763.008,A 0.000,B 0.000,C 90.000,E1 181.489} C_DIS
LIN {X 0.003,Y -141.306,Z 762.972,A 0.000,B 0.000,C 90.000,E1 174.951} C_DIS
LIN {X -0.039,Y -142.667,Z 762.956,A 0.000,B 0.000,C 90.000,E1 172.186} C_DIS
LIN {X 0.083,Y -145.015,Z 762.931,A 0.000,B 0.000,C 90.000,E1 167.521} C_DIS
LIN {X 0.041,Y -147.642,Z 762.910,A 0.000,B 0.000,C 90.000,E1 163.866} C_DIS
LIN {X -0.024,Y -150.274,Z 762.890,A 0.000,B 0.000,C 90.000,E1 160.242} C_DIS
LIN {X -0.011,Y -153.676,Z 762.870,A 0.000,B 0.000,C 90.000,E1 156.613} C_DIS
LIN {X 0.045,Y -157.091,Z 762.850,A 0.000,B 0.000,C 90.000,E1 152.999} C_DIS
LIN {X -0.016,Y -161.228,Z 762.830,A 0.000,B 0.000,C 90.000,E1 149.459} C_DIS
LIN {X 0.069,Y -163.316,Z 762.820,A 0.000,B 0.000,C 90.000,E1 147.661} C_DIS
LIN {X -0.060,Y -167.767,Z 762.801,A 0.000,B 0.000,C 90.000,E1 144.196} C_DIS
LIN {X 0.092,Y -171.583,Z 762.786,A 0.000,B 0.000,C 90.000,E1 141.537} C_DIS
LIN {X -0.108,Y -176.532,Z 762.767,A 0.000,B 0.000,C 90.000,E1 138.162} C_DIS
LIN {X 0.016,Y -180.831,Z 762.753,A 0.000,B 0.000,C 90.000,E1 135.567} C_DIS
LIN {X 0.000,Y -186.242,Z 762.734,A 0.000,B 0.000,C 90.000,E1 132.204} C_DIS
LIN {X 0.058,Y -191.348,Z 762.719,A 0.000,B 0.000,C 90.000,E1 129.402} C_DIS
LIN {X -0.060,Y -192.216,Z 762.716,A 0.000,B 0.000,C 90.000,E1 128.910} C_DIS
LIN {X -0.125,Y -291.948,Z 762.716,A 0.000,B 0.000,C 90.000,E1 128.910} C_DIS
LIN {X 0.117,Y -295.768,Z 762.715,A 0.000,B 0.000,C 90.000,E1 128.749} C_DIS
LIN {X 0.131,Y -298.876,Z 762.714,A 0.000,B 0.000,C 90.000,E1 128.543} C_DIS
LIN {X -0.025,Y -302.559,Z 762.712,A 0.000,B 0.000,C 90.000,E1 128.177} C_DIS
LIN {X -0.097,Y -304.502,Z 762.710,A 0.000,B 0.000,C 90.000,E1 127.890} C_DIS
LIN {X 0.018,Y -306.032,Z 762.709,A 0.000,B 0.000,C 90.000,E1 127.569} C_DIS
LIN {X 0.038,Y -307.362,Z 762.707,A 0.000,B 0.000,C 90.000,E1 127.237} C_DIS
LIN {X 0.139,Y -315.160,Z 762.692,A 0.000,B 0.000,C 90.000,E1 124.612} C_DIS
LIN {X -0.176,Y -326.092,Z 762.675,A 0.000,B 0.000,C 90.000,E1 121.465} C_DIS
LIN {X -0.062,Y -337.314,Z 762.659,A 0.000,B 0.000,C 90.000,E1 118.615} C_DIS
LIN {X -0.101,Y -349.949,Z 762.643,A 0.000,B 0.000,C 90.000,E1 115.848} C_DIS
LIN {X 0.181,Y -362.460,Z 762.630,A 0.000,B 0.000,C 90.000,E1 113.387} C_DIS
LIN {X 0.025,Y -376.268,Z 762.617,A 0.000,B 0.000,C 90.000,E1 111.046} C_DIS
LIN {X 0.079,Y -391.470,Z 762.604,A 0.000,B 0.000,C 90.000,E1 108.725} C_DIS
LIN {X -0.123,Y -408.178,Z 762.592,A 0.000,B 0.000,C 90.000,E1 106.496} C_DIS
LIN {X -0.157,Y -426.512,Z 762.579,A 0.000,B 0.000,C 90.000,E1 104.300} C_DIS
LIN {X -0.036,Y -446.304,Z 762.568,A 0.000,B 0.000,C 90.000,E1 102.175} C_DIS
LIN {X -0.190,Y -466.734,Z 762.557,A 0.000,B 0.000,C 90.000,E1 100.254} C_DIS
LIN {X -0.163,Y -469.096,Z 762.556,A 0.000,B 0.000,C 90.000,E1 100.018} C_DIS
LIN {X 0.220,Y -470.964,Z 762.554,A 0.000,B 0.000,C 90.000,E1 99.726} C_DIS
LIN {X 0.062,Y -472.380,Z 762.553,A 0.000,B 0.000,C 90.000,E1 99.500} C_DIS
LIN {X 0.242,Y -474.260,Z 762.550,A 0.000,B 0.000,C 90.000,E1 98.973} C_DIS
LIN {X -0.115,Y -475.035,Z 762.547,A 0.000,B 0.000,C 90.000,E1 98.511} C_DIS
LIN {X 0.012,Y -474.839,Z 762.544,A 0.000,B 0.000,C 90.000,E1 97.992} C_DIS
LIN {X 0.145,Y -473.646,Z 762.542,A 0.000,B 0.000,C 90.000,E1 97.473} C_DIS
LIN {X 0.006,Y -472.622,Z 762.540,A 0.000,B 0.000,C 90.000,E1 97.239} C_DIS
LIN {X -0.134,Y -471.244,Z 762.539,A 0.000,B 0.000,C 90.000,E1 97.004} C_DIS
LIN {X 0.229,Y -451.877,Z 762.522,A 0.000,B 0.000,C 90.000,E1 93.898} C_DIS
LIN {X -0.138,Y -441.427,Z 762.512,A 0.000,B 0.000,C 90.000,E1 92.121} C_DIS
LIN {X 0.019,Y -432.332,Z 762.503,A 0.000,B 0.000,C 90.000,E1 90.516} C_DIS
LIN {X 0.005,Y -422.843,Z 762.494,A 0.000,B 0.000,C 90.000,E1 88.912} C_DIS
LIN {X -0.074,Y -411.695,Z 762.483,A 0.000,B 0.000,C 90.000,E1 87.020} C_DIS
LIN {X 0.071,Y -400.420,Z 762.473,A 0.000,B 0.000,C 90.000,E1 85.065} C_DIS
LIN {X 0.034,Y -387.524,Z 762.460,A 0.000,B 0.000,C 90.000,E1 82.818} C_DIS
LIN {X 0.123,Y -371.931,Z 762.444,A 0.000,B 0.000,C 90.000,E1 79.926} C_DIS
LIN {X -0.027,Y -355.629,Z 762.426,A 0.000,B 0.000,C 90.000,E1 76.700} C_DIS
LIN {X -0.020,Y -344.229,Z 762.413,A 0.000,B 0.000,C 90.000,E1 74.283} C_DIS
LIN {X -0.014,Y -332.977,Z 762.399,A 0.000,B 0.000,C 90.000,E1 71.819} C_DIS
LIN {X 0.080,Y -320.794,Z 762.383,A 0.000,B 0.000,C 90.000,E1 68.975} C_DIS
LIN {X -0.167,Y -306.871,Z 762.364,A 0.000,B 0.000,C 90.000,E1 65.485} C_DIS
LIN {X 0.059,Y -295.402,Z 762.345,A 0.000,B 0.000,C 90.000,E1 62.153} C_DIS
LIN {X 0.117,Y -284.927,Z 762.327,A 0.000,B 0.000,C 90.000,E1 58.791} C_DIS
LIN {X 0.004,Y -277.076,Z 762.312,A 0.000,B 0.000,C 90.000,E1 56.087} C_DIS
LIN {X -0.068,Y -269.365,Z 762.296,A 0.000,B 0.000,C 90.000,E1 53.336} C_DIS
LIN {X -0.140,Y -263.610,Z 762.285,A 0.000,B 0.000,C 90.000,E1 51.251} C_DIS
LIN {X -0.100,Y -255.958,Z 762.269,A 0.000,B 0.000,C 90.000,E1 48.405} C_DIS
LIN {X 0.064,Y -248.268,Z 762.253,A 0.000,B 0.000,C 90.000,E1 45.486} C_DIS
LIN {X 0.054,Y -242.588,Z 762.241,A 0.000,B 0.000,C 90.000,E1 43.299} C_DIS
LIN {X 0.076,Y -235.034,Z 762.224,A 0.000,B 0.000,C 90.000,E1 40.334} C_DIS
LIN {X 0.027,Y -226.010,Z 762.203,A 0.000,B 0.000,C 90.000,E1 36.583} C_DIS
LIN {X 0.115,Y -219.198,Z 762.186,A 0.000,B 0.000,C 90.000,E1 33.499} C_DIS
LIN {X 0.045,Y -212.999,Z 762.169,A 0.000,B 0.000,C 90.000,E1 30.413} C_DIS
LIN {X 0.085,Y -207.459,Z 762.152,A 0.000,B 0.000,C 90.000,E1 27.257} C_DIS
LIN {X -0.128,Y -201.604,Z 762.129,A 0.000,B 0.000,C 90.000,E1 23.334} C_DIS
LIN {X -0.010,Y -196.813,Z 762.107,A 0.000,B 0.000,C 90.000,E1 19.268} C_DIS
LIN {X 0.009,Y -193.150,Z 762.084,A 0.000,B 0.000,C 90.000,E1 15.190} C_DIS
LIN {X 0.034,Y -190.074,Z 762.057,A 0.000,B 0.000,C 90.000,E1 10.254} C_DIS
LIN {X -0.071,Y -190.710,Z 761.961,A 0.000,B 0.000,C 90.000,E1 352.932} C_DIS
LIN {X -0.070,Y -193.999,Z 761.933,A 0.000,B 0.000,C 90.000,E1 347.993} C_DIS
LIN {X 0.077,Y -197.891,Z 761.910,A 0.000,B 0.000,C 90.000,E1 343.866} C_DIS
LIN {X 0.049,Y -202.827,Z 761.888,A 0.000,B 0.000,C 90.000,E1 339.826} C_DIS
LIN {X -0.029,Y -208.687,Z 761.866,A 0.000,B 0.000,C 90.000,E1 335.845} C_DIS
LIN {X -0.038,Y -215.368,Z 761.844,A 0.000,B 0.000,C 90.000,E1 331.897} C_DIS
LIN {X -0.003,Y -222.857,Z 761.822,A 0.000,B 0.000,C 90.000,E1 327.995} C_DIS
LIN {X -0.135,Y -230.878,Z 761.801,A 0.000,B 0.000,C 90.000,E1 324.196} C_DIS
LIN {X -0.019,Y -239.655,Z 761.780,A 0.000,B 0.000,C 90.000,E1 320.400} C_DIS
LIN {X -0.023,Y -249.205,Z 761.759,A 0.000,B 0.000,C 90.000,E1 316.701} C_DIS
LIN {X -0.087,Y -259.737,Z 761.739,A 0.000,B 0.000,C 90.000,E1 313.095} C_DIS
LIN {X 0.054,Y -271.177,Z 761.720,A 0.000,B 0.000,C 90.000,E1 309.519} C_DIS
LIN {X -0.127,Y -283.793,Z 761.700,A 0.000,B 0.000,C 90.000,E1 306.091} C_DIS
LIN {X -0.106,Y -294.827,Z 761.685,A 0.000,B 0.000,C 90.000,E1 303.372} C_DIS
LIN {X 0.111,Y -305.626,Z 761.672,A 0.000,B 0.000,C 90.000,E1 301.003} C_DIS
LIN {X 0.048,Y -322.878,Z 761.654,A 0.000,B 0.000,C 90.000,E1 297.769} C_DIS
LIN {X -0.163,Y -335.776,Z 761.642,A 0.000,B 0.000,C 90.000,E1 295.591} C_DIS
LIN {X 0.124,Y -353.726,Z 761.627,A 0.000,B 0.000,C 90.000,E1 292.770} C_DIS
LIN {X -0.046,Y -375.489,Z 761.610,A 0.000,B 0.000,C 90.000,E1 289.812} C_DIS
LIN {X 0.083,Y -399.459,Z 761.594,A 0.000,B 0.000,C 90.000,E1 286.913} C_DIS
LIN {X -0.085,Y -411.755,Z 761.586,A 0.000,B 0.000,C 90.000,E1 285.536} C_DIS
LIN {X 0.231,Y -423.713,Z 761.579,A 0.000,B 0.000,C 90.000,E1 284.120} C_DIS
LIN {X -0.203,Y -435.382,Z 761.571,A 0.000,B 0.000,C 90.000,E1 282.827} C_DIS
LIN {X 0.174,Y -444.473,Z 761.565,A 0.000,B 0.000,C 90.000,E1 281.715} C_DIS
LIN {X 0.227,Y -453.000,Z 761.559,A 0.000,B 0.000,C 90.000,E1 280.658} C_DIS
LIN {X 0.124,Y -463.057,Z 761.552,A 0.000,B 0.000,C 90.000,E1 279.378} C_DIS
LIN {X -0.223,Y -470.795,Z 761.547,A 0.000,B 0.000,C 90.000,E1 278.398} C_DIS
LIN {X 0.053,Y -477.858,Z 761.541,A 0.000,B 0.000,C 90.000,E1 277.352} C_DIS
LIN {X 0.002,Y -482.449,Z 761.537,A 0.000,B 0.000,C 90.000,E1 276.606} C_DIS
LIN {X 0.050,Y -486.260,Z 761.533,A 0.000,B 0.000,C 90.000,E1 275.853} C_DIS
LIN {X -0.122,Y -487.388,Z 761.531,A 0.000,B 0.000,C 90.000,E1 275.625} C_DIS
LIN {X 0.078,Y -489.320,Z 761.528,A 0.000,B 0.000,C 90.000,E1 275.106} C_DIS
LIN {X -0.204,Y -490.895,Z 761.526,A 0.000,B 0.000,C 90.000,E1 274.645} C_DIS
LIN {X -0.024,Y -492.071,Z 761.523,A 0.000,B 0.000,C 90.000,E1 274.131} C_DIS
LIN {X 0.203,Y -492.876,Z 761.520,A 0.000,B 0.000,C 90.000,E1 273.612} C_DIS
LIN {X -0.088,Y -493.277,Z 761.517,A 0.000,B 0.000,C 90.000,E1 273.154} C_DIS
LIN {X 0.147,Y -493.274,Z 761.515,A 0.000,B 0.000,C 90.000,E1 272.636} C_DIS
LIN {X -0.134,Y -492.801,Z 761.512,A 0.000,B 0.000,C 90.000,E1 272.178} C_DIS
LIN {X 0.095,Y -491.886,Z 761.509,A 0.000,B 0.000,C 90.000,E1 271.661} C_DIS
LIN {X -0.185,Y -490.447,Z 761.507,A 0.000,B 0.000,C 90.000,E1 271.203} C_DIS
LIN {X 0.020,Y -488.508,Z 761.504,A 0.000,B 0.000,C 90.000,E1 270.688} C_DIS
LIN {X -0.125,Y -487.375,Z 761.502,A 0.000,B 0.000,C 90.000,E1 270.458} C_DIS
LIN {X 0.064,Y -484.521,Z 761.500,A 0.000,B 0.000,C 90.000,E1 269.943} C_DIS
LIN {X 0.233,Y -480.985,Z 761.497,A 0.000,B 0.000,C 90.000,E1 269.427} C_DIS
LIN {X -0.097,Y -476.648,Z 761.494,A 0.000,B 0.000,C 90.000,E1 268.969} C_DIS
LIN {X 0.088,Y -471.427,Z 761.491,A 0.000,B 0.000,C 90.000,E1 268.453} C_DIS
LIN {X -0.033,Y -468.472,Z 761.490,A 0.000,B 0.000,C 90.000,E1 268.224} C_DIS
LIN {X 0.161,Y -462.193,Z 761.488,A 0.000,B 0.000,C 90.000,E1 267.764} C_DIS
LIN {X 0.046,Y -459.054,Z 761.487,A 0.000,B 0.000,C 90.000,E1 267.593} C_DIS
LIN {X 0.110,Y -452.028,Z 761.485,A 0.000,B 0.000,C 90.000,E1 267.249} C_DIS
LIN {X -0.204,Y -444.694,Z 761.483,A 0.000,B 0.000,C 90.000,E1 267.020} C_DIS
LIN {X -0.017,Y -436.449,Z 761.482,A 0.000,B 0.000,C 90.000,E1 266.788} C_DIS
LIN {X 0.179,Y -427.403,Z 761.481,A 0.000,B 0.000,C 90.000,E1 266.617} C_DIS
LIN {X 0.172,Y -420.081,Z 761.481,A 0.000,B 0.000,C 90.000,E1 266.560} C_DIS
LIN {X 0.049,Y -180.954,Z 761.481,A 0.000,B 0.000,C 90.000,E1 266.560} C_DIS
LIN {X -0.008,Y -180.816,Z 761.471,A 0.000,B 0.000,C 90.000,E1 264.837} C_DIS
LIN {X 0.069,Y -178.919,Z 761.443,A 0.000,B 0.000,C 90.000,E1 259.746} C_DIS
LIN {X -0.023,Y -175.964,Z 761.415,A 0.000,B 0.000,C 90.000,E1 254.685} C_DIS
LIN {X 0.094,Y -175.442,Z 761.410,A 0.000,B 0.000,C 90.000,E1 253.795} C_DIS
LIN {X -0.066,Y -172.198,Z 761.386,A 0.000,B 0.000,C 90.000,E1 249.571} C_DIS
LIN {X -0.088,Y -171.672,Z 761.382,A 0.000,B 0.000,C 90.000,E1 248.720} C_DIS
LIN {X -0.096,Y -167.898,Z 761.358,A 0.000,B 0.000,C 90.000,E1 244.409} C_DIS
LIN {X 0.070,Y -166.637,Z 761.348,A 0.000,B 0.000,C 90.000,E1 242.615} C_DIS
LIN {X -0.023,Y -162.622,Z 761.324,A 0.000,B 0.000,C 90.000,E1 238.280} C_DIS
LIN {X 0.037,Y -161.308,Z 761.314,A 0.000,B 0.000,C 90.000,E1 236.501} C_DIS
LIN {X -0.053,Y -157.305,Z 761.289,A 0.000,B 0.000,C 90.000,E1 232.110} C_DIS
LIN {X 0.099,Y -155.283,Z 761.275,A 0.000,B 0.000,C 90.000,E1 229.380} C_DIS
LIN {X 0.027,Y -151.647,Z 761.250,A 0.000,B 0.000,C 90.000,E1 224.919} C_DIS
LIN {X -0.036,Y -150.515,Z 761.240,A 0.000,B 0.000,C 90.000,E1 223.137} C_DIS
LIN {X -0.013,Y -147.239,Z 761.214,A 0.000,B 0.000,C 90.000,E1 218.588} C_DIS
LIN {X -0.047,Y -145.264,Z 761.194,A 0.000,B 0.000,C 90.000,E1 214.945} C_DIS
LIN {X -0.013,Y -142.374,Z 761.163,A 0.000,B 0.000,C 90.000,E1 209.411} C_DIS
LIN {X 0.037,Y -141.349,Z 761.148,A 0.000,B 0.000,C 90.000,E1 206.616} C_DIS
LIN {X 0.020,Y -139.338,Z 761.112,A 0.000,B 0.000,C 90.000,E1 200.120} C_DIS
LIN {X 0.070,Y -139.005,Z 761.101,A 0.000,B 0.000,C 90.000,E1 198.236} C_DIS
LIN {X 0.026,Y -138.339,Z 761.055,A 0.000,B 0.000,C 90.000,E1 189.849} C_DIS
LIN {X 0.049,Y -139.406,Z 761.008,A 0.000,B 0.000,C 90.000,E1 181.432} C_DIS
LIN {X -0.038,Y -141.314,Z 760.972,A 0.000,B 0.000,C 90.000,E1 174.951} C_DIS
LIN {X 0.060,Y -142.673,Z 760.956,A 0.000,B 0.000,C 90.000,E1 172.129} C_DIS
LIN {X 0.041,Y -145.025,Z 760.931,A 0.000,B 0.000,C 90.000,E1 167.521} C_DIS
LIN {X -0.001,Y -147.652,Z 760.910,A 0.000,B 0.000,C 90.000,E1 163.866} C_DIS
LIN {X -0.067,Y -150.288,Z 760.890,A 0.000,B 0.000,C 90.000,E1 160.242} C_DIS
LIN {X -0.054,Y -153.694,Z 760.870,A 0.000,B 0.000,C 90.000,E1 156.613} C_DIS
LIN {X 0.001,Y -157.108,Z 760.850,A 0.000,B 0.000,C 90.000,E1 152.999} C_DIS
LIN {X -0.061,Y -161.249,Z 760.830,A 0.000,B 0.000,C 90.000,E1 149.459} C_DIS
LIN {X 0.024,Y -163.334,Z 760.820,A 0.000,B 0.000,C 90.000,E1 147.661} C_DIS
LIN {X 0.030,Y -167.789,Z 760.801,A 0.000,B 0.000,C 90.000,E1 144.149} C_DIS
LIN {X 0.046,Y -171.604,Z 760.786,A 0.000,B 0.000,C 90.000,E1 141.537} C_DIS
LIN {X 0.093,Y -176.557,Z 760.767,A 0.000,B 0.000,C 90.000,E1 138.081} C_DIS
LIN {X -0.032,Y -180.856,Z 760.753,A 0.000,B 0.000,C 90.000,E1 135.567} C_DIS
LIN {X -0.049,Y -186.267,Z 760.734,A 0.000,B 0.000,C 90.000,E1 132.204} C_DIS
LIN {X 0.015,Y -191.369,Z 760.719,A 0.000,B 0.000,C 90.000,E1 129.402} C_DIS
LIN {X 0.013,Y -192.179,Z 760.716,A 0.000,B 0.000,C 90.000,E1 128.910} C_DIS
LIN {X -0.016,Y -291.487,Z 760.716,A 0.000,B 0.000,C 90.000,E1 128.910} C_DIS
LIN {X 0.178,Y -293.789,Z 760.716,A 0.000,B 0.000,C 90.000,E1 128.830} C_DIS
LIN {X 0.013,Y -297.164,Z 760.715,A 0.000,B 0.000,C 90.000,E1 128.705} C_DIS
LIN {X 0.178,Y -300.604,Z 760.713,A 0.000,B 0.000,C 90.000,E1 128.382} C_DIS
LIN {X -0.071,Y -304.243,Z 760.711,A 0.000,B 0.000,C 90.000,E1 127.935} C_DIS
LIN {X -0.065,Y -305.952,Z 760.709,A 0.000,B 0.000,C 90.000,E1 127.604} C_DIS
LIN {X 0.130,Y -307.293,Z 760.707,A 0.000,B 0.000,C 90.000,E1 127.237} C_DIS
LIN {X -0.106,Y -318.201,Z 760.687,A 0.000,B 0.000,C 90.000,E1 123.706} C_DIS
LIN {X 0.117,Y -328.384,Z 760.671,A 0.000,B 0.000,C 90.000,E1 120.797} C_DIS
LIN {X 0.149,Y -339.901,Z 760.656,A 0.000,B 0.000,C 90.000,E1 117.975} C_DIS
LIN {X 0.190,Y -352.859,Z 760.640,A 0.000,B 0.000,C 90.000,E1 115.207} C_DIS
LIN {X 0.073,Y -365.678,Z 760.627,A 0.000,B 0.000,C 90.000,E1 112.823} C_DIS
LIN {X -0.010,Y -379.816,Z 760.614,A 0.000,B 0.000,C 90.000,E1 110.482} C_DIS
LIN {X -0.003,Y -395.375,Z 760.601,A 0.000,B 0.000,C 90.000,E1 108.181} C_DIS
LIN {X -0.116,Y -412.467,Z 760.589,A 0.000,B 0.000,C 90.000,E1 105.953} C_DIS
LIN {X -0.153,Y -431.217,Z 760.576,A 0.000,B 0.000,C 90.000,E1 103.772} C_DIS
LIN {X 0.174,Y -451.217,Z 760.565,A 0.000,B 0.000,C 90.000,E1 101.658} C_DIS
LIN {X -0.106,Y -466.588,Z 760.557,A 0.000,B 0.000,C 90.000,E1 100.254} C_DIS
LIN {X -0.059,Y -468.961,Z 760.556,A 0.000,B 0.000,C 90.000,E1 100.018} C_DIS
LIN {X -0.092,Y -470.762,Z 760.554,A 0.000,B 0.000,C 90.000,E1 99.792} C_DIS
LIN {X -0.240,Y -472.271,Z 760.553,A 0.000,B 0.000,C 90.000,E1 99.557} C_DIS
LIN {X 0.077,Y -473.400,Z 760.552,A 0.000,B 0.000,C 90.000,E1 99.265} C_DIS
LIN {X 0.189,Y -474.747,Z 760.549,A 0.000,B 0.000,C 90.000,E1 98.746} C_DIS
LIN {X -0.089,Y -475.075,Z 760.546,A 0.000,B 0.000,C 90.000,E1 98.276} C_DIS
LIN {X 0.038,Y -474.439,Z 760.543,A 0.000,B 0.000,C 90.000,E1 97.757} C_DIS
LIN {X 0.169,Y -472.740,Z 760.540,A 0.000,B 0.000,C 90.000,E1 97.239} C_DIS
LIN {X 0.028,Y -471.397,Z 760.539,A 0.000,B 0.000,C 90.000,E1 97.004} C_DIS
LIN {X -0.060,Y -452.032,Z 760.522,A 0.000,B 0.000,C 90.000,E1 93.955} C_DIS
LIN {X 0.026,Y -441.585,Z 760.512,A 0.000,B 0.000,C 90.000,E1 92.121} C_DIS
LIN {X 0.184,Y -432.503,Z 760.503,A 0.000,B 0.000,C 90.000,E1 90.516} C_DIS
LIN {X 0.168,Y -423.034,Z 760.494,A 0.000,B 0.000,C 90.000,E1 88.912} C_DIS
LIN {X 0.084,Y -411.881,Z 760.484,A 0.000,B 0.000,C 90.000,E1 87.020} C_DIS
LIN {X -0.165,Y -400.635,Z 760.473,A 0.000,B 0.000,C 90.000,E1 85.122} C_DIS
LIN {X 0.197,Y -387.736,Z 760.460,A 0.000,B 0.000,C 90.000,E1 82.818} C_DIS
LIN {X -0.080,Y -372.162,Z 760.444,A 0.000,B 0.000,C 90.000,E1 79.982} C_DIS
LIN {X 0.132,Y -355.846,Z 760.426,A 0.000,B 0.000,C 90.000,E1 76.700} C_DIS
LIN {X 0.139,Y -344.433,Z 760.413,A 0.000,B 0.000,C 90.000,E1 74.283} C_DIS
LIN {X 0.145,Y -333.202,Z 760.399,A 0.000,B 0.000,C 90.000,E1 71.819} C_DIS
LIN {X -0.056,Y -321.041,Z 760.383,A 0.000,B 0.000,C 90.000,E1 69.028} C_DIS
LIN {X -0.007,Y -307.146,Z 760.364,A 0.000,B 0.000,C 90.000,E1 65.485} C_DIS
LIN {X 0.092,Y -294.653,Z 760.344,A 0.000,B 0.000,C 90.000,E1 61.847} C_DIS
LIN {X -0.120,Y -284.299,Z 760.325,A 0.000,B 0.000,C 90.000,E1 58.535} C_DIS
LIN {X -0.096,Y -276.497,Z 760.310,A 0.000,B 0.000,C 90.000,E1 55.801} C_DIS
LIN {X 0.038,Y -268.860,Z 760.294,A 0.000,B 0.000,C 90.000,E1 53.004} C_DIS
LIN {X 0.115,Y -263.138,Z 760.283,A 0.000,B 0.000,C 90.000,E1 50.884} C_DIS
LIN {X -0.058,Y -255.493,Z 760.267,A 0.000,B 0.000,C 90.000,E1 48.081} C_DIS
LIN {X 0.096,Y -247.820,Z 760.251,A 0.000,B 0.000,C 90.000,E1 45.162} C_DIS
LIN {X -0.090,Y -242.137,Z 760.239,A 0.000,B 0.000,C 90.000,E1 43.014} C_DIS
LIN {X 0.083,Y -234.582,Z 760.222,A 0.000,B 0.000,C 90.000,E1 40.011} C_DIS
LIN {X -0.125,Y -225.572,Z 760.201,A 0.000,B 0.000,C 90.000,E1 36.297} C_DIS
LIN {X -0.044,Y -218.786,Z 760.184,A 0.000,B 0.000,C 90.000,E1 33.214} C_DIS
LIN {X 0.059,Y -212.643,Z 760.167,A 0.000,B 0.000,C 90.000,E1 30.079} C_DIS
LIN {X -0.006,Y -207.171,Z 760.150,A 0.000,B 0.000,C 90.000,E1 26.950} C_DIS
LIN {X -0.023,Y -202.460,Z 760.132,A 0.000,B 0.000,C 90.000,E1 23.770} C_DIS
LIN {X -0.065,Y -197.509,Z 760.110,A 0.000,B 0.000,C 90.000,E1 19.758} C_DIS
LIN {X 0.033,Y -193.715,Z 760.087,A 0.000,B 0.000,C 90.000,E1 15.662} C_DIS
LIN {X -0.108,Y -190.479,Z 760.060,A 0.000,B 0.000,C 90.000,E1 10.782} C_DIS
LIN {X 0.057,Y -188.339,Z 760.014,A 0.000,B 0.000,C 90.000,E1 2.465} C_DIS
LIN {X -0.013,Y -190.406,Z 759.965,A 0.000,B 0.000,C 90.000,E1 353.742} C_DIS
LIN {X -0.059,Y -193.452,Z 759.938,A 0.000,B 0.000,C 90.000,E1 348.814} C_DIS
LIN {X 0.021,Y -197.173,Z 759.915,A 0.000,B 0.000,C 90.000,E1 344.700} C_DIS
LIN {X 0.009,Y -200.824,Z 759.897,A 0.000,B 0.000,C 90.000,E1 341.456} C_DIS
LIN {X 0.098,Y -206.346,Z 759.875,A 0.000,B 0.000,C 90.000,E1 337.411} C_DIS
LIN {X 0.023,Y -212.681,Z 759.853,A 0.000,B 0.000,C 90.000,E1 333.461} C_DIS
LIN {X 0.051,Y -219.877,Z 759.831,A 0.000,B 0.000,C 90.000,E1 329.537} C_DIS
LIN {X 0.082,Y -227.687,Z 759.809,A 0.000,B 0.000,C 90.000,E1 325.674} C_DIS
LIN {X -0.006,Y -236.119,Z 759.788,A 0.000,B 0.000,C 90.000,E1 321.904} C_DIS
LIN {X 0.062,Y -245.283,Z 759.768,A 0.000,B 0.000,C 90.000,E1 318.162} C_DIS
LIN {X 0.032,Y -254.373,Z 759.749,A 0.000,B 0.000,C 90.000,E1 314.879} C_DIS
LIN {X -0.032,Y -265.314,Z 759.729,A 0.000,B 0.000,C 90.000,E1 311.310} C_DIS
LIN {X -0.061,Y -277.325,Z 759.710,A 0.000,B 0.000,C 90.000,E1 307.810} C_DIS
LIN {X -0.168,Y -290.536,Z 759.691,A 0.000,B 0.000,C 90.000,E1 304.405} C_DIS
LIN {X 0.101,Y -300.842,Z 759.678,A 0.000,B 0.000,C 90.000,E1 302.005} C_DIS
LIN {X -0.122,Y -312.334,Z 759.665,A 0.000,B 0.000,C 90.000,E1 299.745} C_DIS
LIN {X 0.157,Y -330.176,Z 759.647,A 0.000,B 0.000,C 90.000,E1 296.488} C_DIS
LIN {X -0.033,Y -345.471,Z 759.633,A 0.000,B 0.000,C 90.000,E1 294.027} C_DIS
LIN {X 0.145,Y -366.429,Z 759.617,A 0.000,B 0.000,C 90.000,E1 290.972} C_DIS
LIN {X -0.026,Y -387.070,Z 759.602,A 0.000,B 0.000,C 90.000,E1 288.362} C_DIS
LIN {X -0.121,Y -404.230,Z 759.591,A 0.000,B 0.000,C 90.000,E1 286.386} C_DIS
LIN {X 0.184,Y -416.327,Z 759.583,A 0.000,B 0.000,C 90.000,E1 284.954} C_DIS
LIN {X 0.172,Y -428.169,Z 759.576,A 0.000,B 0.000,C 90.000,E1 283.592} C_DIS
LIN {X -0.200,Y -439.727,Z 759.568,A 0.000,B 0.000,C 90.000,E1 282.299} C_DIS
LIN {X -0.209,Y -448.553,Z 759.562,A 0.000,B 0.000,C 90.000,E1 281.243} C_DIS
LIN {X 0.068,Y -458.837,Z 759.555,A 0.000,B 0.000,C 90.000,E1 279.905} C_DIS
LIN {X 0.040,Y -468.693,Z 759.548,A 0.000,B 0.000,C 90.000,E1 278.624} C_DIS
LIN {X -0.243,Y -475.978,Z 759.542,A 0.000,B 0.000,C 90.000,E1 277.644} C_DIS
LIN {X 0.227,Y -480.870,Z 759.538,A 0.000,B 0.000,C 90.000,E1 276.834} C_DIS
LIN {X 0.206,Y -484.954,Z 759.534,A 0.000,B 0.000,C 90.000,E1 276.087} C_DIS
LIN {X -0.091,Y -487.296,Z 759.531,A 0.000,B 0.000,C 90.000,E1 275.625} C_DIS
LIN {X 0.109,Y -489.269,Z 759.528,A 0.000,B 0.000,C 90.000,E1 275.106} C_DIS
LIN {X -0.173,Y -490.871,Z 759.526,A 0.000,B 0.000,C 90.000,E1 274.645} C_DIS
LIN {X 0.007,Y -492.107,Z 759.523,A 0.000,B 0.000,C 90.000,E1 274.131} C_DIS
LIN {X 0.233,Y -492.928,Z 759.520,A 0.000,B 0.000,C 90.000,E1 273.612} C_DIS
LIN {X -0.057,Y -493.343,Z 759.518,A 0.000,B 0.000,C 90.000,E1 273.154} C_DIS
LIN {X 0.177,Y -493.307,Z 759.515,A 0.000,B 0.000,C 90.000,E1 272.636} C_DIS
LIN {X -0.102,Y -492.864,Z 759.512,A 0.000,B 0.000,C 90.000,E1 272.178} C_DIS
LIN {X 0.128,Y -491.982,Z 759.509,A 0.000,B 0.000,C 90.000,E1 271.661} C_DIS
LIN {X -0.154,Y -490.584,Z 759.507,A 0.000,B 0.000,C 90.000,E1 271.203} C_DIS
LIN {X 0.052,Y -488.686,Z 759.504,A 0.000,B 0.000,C 90.000,E1 270.688} C_DIS
LIN {X -0.237,Y -486.207,Z 759.501,A 0.000,B 0.000,C 90.000,E1 270.229} C_DIS
LIN {X -0.056,Y -483.070,Z 759.498,A 0.000,B 0.000,C 90.000,E1 269.714} C_DIS
LIN {X 0.107,Y -479.166,Z 759.496,A 0.000,B 0.000,C 90.000,E1 269.198} C_DIS
LIN {X -0.228,Y -474.421,Z 759.493,A 0.000,B 0.000,C 90.000,E1 268.740} C_DIS
LIN {X 0.100,Y -471.727,Z 759.491,A 0.000,B 0.000,C 90.000,E1 268.453} C_DIS
LIN {X 0.078,Y -465.776,Z 759.489,A 0.000,B 0.000,C 90.000,E1 267.993} C_DIS
LIN {X 0.067,Y -459.353,Z 759.487,A 0.000,B 0.000,C 90.000,E1 267.593} C_DIS
LIN {X 0.116,Y -452.372,Z 759.485,A 0.000,B 0.000,C 90.000,E1 267.249} C_DIS
LIN {X -0.230,Y -444.909,Z 759.483,A 0.000,B 0.000,C 90.000,E1 267.020} C_DIS
LIN {X -0.072,Y -436.707,Z 759.482,A 0.000,B 0.000,C 90.000,E1 266.788} C_DIS
LIN {X 0.107,Y -427.649,Z 759.481,A 0.000,B 0.000,C 90.000,E1 266.617} C_DIS
LIN {X 0.097,Y -420.453,Z 759.481,A 0.000,B 0.000,C 90.000,E1 266.560} C_DIS
LIN {X 0.038,Y -416.736,Z 759.481,A 0.000,B 0.000,C 90.000,E1 266.560} C_DIS
LIN {X -0.009,Y -180.953,Z 759.481,A 0.000,B 0.000,C 90.000,E1 266.560} C_DIS
LIN {X -0.044,Y -180.813,Z 759.471,A 0.000,B 0.000,C 90.000,E1 264.837} C_DIS
LIN {X 0.033,Y -178.914,Z 759.443,A 0.000,B 0.000,C 90.000,E1 259.746} C_DIS
LIN {X -0.057,Y -175.959,Z 759.415,A 0.000,B 0.000,C 90.000,E1 254.685} C_DIS
LIN {X 0.059,Y -175.433,Z 759.410,A 0.000,B 0.000,C 90.000,E1 253.795} C_DIS
LIN {X 0.062,Y -172.191,Z 759.386,A 0.000,B 0.000,C 90.000,E1 249.518} C_DIS
LIN {X 0.038,Y -171.664,Z 759.382,A 0.000,B 0.000,C 90.000,E1 248.666} C_DIS
LIN {X 0.021,Y -167.889,Z 759.358,A 0.000,B 0.000,C 90.000,E1 244.357} C_DIS
LIN {X 0.037,Y -166.627,Z 759.348,A 0.000,B 0.000,C 90.000,E1 242.615} C_DIS
LIN {X 0.030,Y -162.613,Z 759.324,A 0.000,B 0.000,C 90.000,E1 238.250} C_DIS
LIN {X 0.004,Y -161.299,Z 759.314,A 0.000,B 0.000,C 90.000,E1 236.501} C_DIS
LIN {X 0.038,Y -157.296,Z 759.289,A 0.000,B 0.000,C 90.000,E1 232.065} C_DIS
LIN {X 0.066,Y -155.271,Z 759.274,A 0.000,B 0.000,C 90.000,E1 229.380} C_DIS
LIN {X -0.005,Y -151.639,Z 759.250,A 0.000,B 0.000,C 90.000,E1 224.919} C_DIS
LIN {X 0.042,Y -150.507,Z 759.240,A 0.000,B 0.000,C 90.000,E1 223.095} C_DIS
LIN {X 0.072,Y -147.233,Z 759.214,A 0.000,B 0.000,C 90.000,E1 218.543} C_DIS
LIN {X 0.041,Y -145.256,Z 759.194,A 0.000,B 0.000,C 90.000,E1 214.898} C_DIS
LIN {X -0.044,Y -142.369,Z 759.163,A 0.000,B 0.000,C 90.000,E1 209.411} C_DIS
LIN {X 0.077,Y -141.754,Z 759.153,A 0.000,B 0.000,C 90.000,E1 207.513} C_DIS
LIN {X 0.004,Y -139.495,Z 759.117,A 0.000,B 0.000,C 90.000,E1 201.046} C_DIS
LIN {X 0.040,Y -139.001,Z 759.101,A 0.000,B 0.000,C 90.000,E1 198.236} C_DIS
LIN {X -0.003,Y -138.338,Z 759.055,A 0.000,B 0.000,C 90.000,E1 189.849} C_DIS
LIN {X 0.019,Y -139.409,Z 759.008,A 0.000,B 0.000,C 90.000,E1 181.432} C_DIS
LIN {X -0.068,Y -141.319,Z 758.972,A 0.000,B 0.000,C 90.000,E1 174.951} C_DIS
LIN {X 0.030,Y -142.678,Z 758.956,A 0.000,B 0.000,C 90.000,E1 172.129} C_DIS
LIN {X 0.010,Y -145.033,Z 758.931,A 0.000,B 0.000,C 90.000,E1 167.521} C_DIS
LIN {X -0.033,Y -147.659,Z 758.910,A 0.000,B 0.000,C 90.000,E1 163.866} C_DIS
LIN {X 0.043,Y -150.297,Z 758.890,A 0.000,B 0.000,C 90.000,E1 160.188} C_DIS
LIN {X -0.086,Y -153.706,Z 758.870,A 0.000,B 0.000,C 90.000,E1 156.613} C_DIS
LIN {X -0.032,Y -157.120,Z 758.850,A 0.000,B 0.000,C 90.000,E1 152.999} C_DIS
LIN {X 0.045,Y -161.264,Z 758.830,A 0.000,B 0.000,C 90.000,E1 149.410} C_DIS
LIN {X -0.028,Y -164.381,Z 758.815,A 0.000,B 0.000,C 90.000,E1 146.786} C_DIS
LIN {X -0.041,Y -169.057,Z 758.796,A 0.000,B 0.000,C 90.000,E1 143.290} C_DIS
LIN {X 0.011,Y -171.618,Z 758.786,A 0.000,B 0.000,C 90.000,E1 141.537} C_DIS
LIN {X 0.059,Y -176.575,Z 758.767,A 0.000,B 0.000,C 90.000,E1 138.081} C_DIS
LIN {X -0.068,Y -180.873,Z 758.753,A 0.000,B 0.000,C 90.000,E1 135.567} C_DIS
LIN {X 0.054,Y -186.287,Z 758.734,A 0.000,B 0.000,C 90.000,E1 132.162} C_DIS
LIN {X -0.017,Y -191.384,Z 758.719,A 0.000,B 0.000,C 90.000,E1 129.402} C_DIS
LIN {X 0.080,Y -192.146,Z 758.716,A 0.000,B 0.000,C 90.000,E1 128.910} C_DIS
LIN {X 0.087,Y -291.517,Z 758.716,A 0.000,B 0.000,C 90.000,E1 128.910} C_DIS
LIN {X 0.123,Y -294.639,Z 758.716,A 0.000,B 0.000,C 90.000,E1 128.830} C_DIS
LIN {X 0.008,Y -297.917,Z 758.715,A 0.000,B 0.000,C 90.000,E1 128.669} C_DIS
LIN {X -0.058,Y -301.498,Z 758.713,A 0.000,B 0.000,C 90.000,E1 128.338} C_DIS
LIN {X -0.169,Y -305.069,Z 758.710,A 0.000,B 0.000,C 90.000,E1 127.810} C_DIS
LIN {X 0.028,Y -306.579,Z 758.708,A 0.000,B 0.000,C 90.000,E1 127.443} C_DIS
LIN {X 0.039,Y -307.767,Z 758.706,A 0.000,B 0.000,C 90.000,E1 127.111} C_DIS
LIN {X -0.179,Y -318.643,Z 758.686,A 0.000,B 0.000,C 90.000,E1 123.579} C_DIS
LIN {X 0.060,Y -328.889,Z 758.670,A 0.000,B 0.000,C 90.000,E1 120.669} C_DIS
LIN {X 0.107,Y -340.473,Z 758.655,A 0.000,B 0.000,C 90.000,E1 117.847} C_DIS
LIN {X 0.162,Y -353.504,Z 758.639,A 0.000,B 0.000,C 90.000,E1 115.079} C_DIS
LIN {X 0.059,Y -366.392,Z 758.626,A 0.000,B 0.000,C 90.000,E1 112.695} C_DIS
LIN {X -0.009,Y -380.604,Z 758.613,A 0.000,B 0.000,C 90.000,E1 110.355} C_DIS
LIN {X 0.014,Y -396.244,Z 758.600,A 0.000,B 0.000,C 90.000,E1 108.055} C_DIS
LIN {X -0.196,Y -413.423,Z 758.588,A 0.000,B 0.000,C 90.000,E1 105.843} C_DIS
LIN {X -0.102,Y -432.268,Z 758.576,A 0.000,B 0.000,C 90.000,E1 103.647} C_DIS
LIN {X -0.147,Y -452.301,Z 758.564,A 0.000,B 0.000,C 90.000,E1 101.591} C_DIS
LIN {X -0.015,Y -467.684,Z 758.556,A 0.000,B 0.000,C 90.000,E1 100.141} C_DIS
LIN {X 0.010,Y -469.822,Z 758.555,A 0.000,B 0.000,C 90.000,E1 99.905} C_DIS
LIN {X 0.034,Y -471.441,Z 758.554,A 0.000,B 0.000,C 90.000,E1 99.670} C_DIS
LIN {X -0.113,Y -472.782,Z 758.552,A 0.000,B 0.000,C 90.000,E1 99.434} C_DIS
LIN {X 0.131,Y -473.775,Z 758.551,A 0.000,B 0.000,C 90.000,E1 99.151} C_DIS
LIN {X -0.150,Y -474.902,Z 758.548,A 0.000,B 0.000,C 90.000,E1 98.681} C_DIS
LIN {X -0.028,Y -475.033,Z 758.545,A 0.000,B 0.000,C 90.000,E1 98.163} C_DIS
LIN {X 0.102,Y -474.195,Z 758.543,A 0.000,B 0.000,C 90.000,E1 97.644} C_DIS
LIN {X -0.236,Y -472.249,Z 758.540,A 0.000,B 0.000,C 90.000,E1 97.182} C_DIS
LIN {X 0.205,Y -467.431,Z 758.536,A 0.000,B 0.000,C 90.000,E1 96.372} C_DIS
LIN {X -0.016,Y -451.438,Z 758.521,A 0.000,B 0.000,C 90.000,E1 93.841} C_DIS
LIN {X 0.061,Y -440.985,Z 758.511,A 0.000,B 0.000,C 90.000,E1 92.007} C_DIS
LIN {X 0.207,Y -431.904,Z 758.502,A 0.000,B 0.000,C 90.000,E1 90.401} C_DIS
LIN {X 0.180,Y -422.426,Z 758.493,A 0.000,B 0.000,C 90.000,E1 88.797} C_DIS
LIN {X 0.082,Y -411.276,Z 758.483,A 0.000,B 0.000,C 90.000,E1 86.906} C_DIS
LIN {X -0.180,Y -400.034,Z 758.472,A 0.000,B 0.000,C 90.000,E1 85.008} C_DIS
LIN {X 0.165,Y -387.149,Z 758.460,A 0.000,B 0.000,C 90.000,E1 82.704} C_DIS
LIN {X -0.069,Y -371.624,Z 758.444,A 0.000,B 0.000,C 90.000,E1 79.859} C_DIS
LIN {X 0.056,Y -355.349,Z 758.426,A 0.000,B 0.000,C 90.000,E1 76.589} C_DIS
LIN {X 0.055,Y -342.528,Z 758.410,A 0.000,B 0.000,C 90.000,E1 73.866} C_DIS
LIN {X 0.017,Y -331.370,Z 758.397,A 0.000,B 0.000,C 90.000,E1 71.402} C_DIS
LIN {X 0.117,Y -318.025,Z 758.379,A 0.000,B 0.000,C 90.000,E1 68.230} C_DIS
LIN {X -0.092,Y -304.463,Z 758.359,A 0.000,B 0.000,C 90.000,E1 64.717} C_DIS
LIN {X 0.068,Y -292.353,Z 758.339,A 0.000,B 0.000,C 90.000,E1 61.051} C_DIS
LIN {X -0.061,Y -282.202,Z 758.321,A 0.000,B 0.000,C 90.000,E1 57.709} C_DIS
LIN {X -0.087,Y -274.490,Z 758.305,A 0.000,B 0.000,C 90.000,E1 54.975} C_DIS
LIN {X 0.152,Y -268.841,Z 758.294,A 0.000,B 0.000,C 90.000,E1 52.844} C_DIS
LIN {X -0.142,Y -263.143,Z 758.282,A 0.000,B 0.000,C 90.000,E1 50.803} C_DIS
LIN {X 0.055,Y -255.500,Z 758.266,A 0.000,B 0.000,C 90.000,E1 47.919} C_DIS
LIN {X 0.015,Y -249.752,Z 758.254,A 0.000,B 0.000,C 90.000,E1 45.769} C_DIS
LIN {X 0.036,Y -244.052,Z 758.242,A 0.000,B 0.000,C 90.000,E1 43.581} C_DIS
LIN {X 0.082,Y -236.461,Z 758.226,A 0.000,B 0.000,C 90.000,E1 40.620} C_DIS
LIN {X 0.072,Y -227.313,Z 758.205,A 0.000,B 0.000,C 90.000,E1 36.870} C_DIS
LIN {X -0.078,Y -218.781,Z 758.184,A 0.000,B 0.000,C 90.000,E1 33.086} C_DIS
LIN {X 0.029,Y -212.647,Z 758.166,A 0.000,B 0.000,C 90.000,E1 29.951} C_DIS
LIN {X -0.035,Y -207.201,Z 758.149,A 0.000,B 0.000,C 90.000,E1 26.821} C_DIS
LIN {X 0.015,Y -201.413,Z 758.127,A 0.000,B 0.000,C 90.000,E1 22.823} C_DIS
LIN {X 0.048,Y -196.705,Z 758.104,A 0.000,B 0.000,C 90.000,E1 18.779} C_DIS
LIN {X 0.058,Y -192.545,Z 758.077,A 0.000,B 0.000,C 90.000,E1 13.883} C_DIS
LIN {X -0.071,Y -189.520,Z 758.045,A 0.000,B 0.000,C 90.000,E1 8.163} C_DIS
LIN {X -0.008,Y -190.514,Z 757.965,A 0.000,B 0.000,C 90.000,E1 353.742} C_DIS
LIN {X -0.050,Y -193.564,Z 757.938,A 0.000,B 0.000,C 90.000,E1 348.814} C_DIS
LIN {X 0.034,Y -197.289,Z 757.915,A 0.000,B 0.000,C 90.000,E1 344.700} C_DIS
LIN {X -0.077,Y -201.960,Z 757.893,A 0.000,B 0.000,C 90.000,E1 340.678} C_DIS
LIN {X -0.075,Y -207.655,Z 757.870,A 0.000,B 0.000,C 90.000,E1 336.666} C_DIS
LIN {X -0.025,Y -214.131,Z 757.848,A 0.000,B 0.000,C 90.000,E1 332.692} C_DIS
LIN {X -0.033,Y -221.488,Z 757.827,A 0.000,B 0.000,C 90.000,E1 328.791} C_DIS
LIN {X -0.143,Y -229.383,Z 757.805,A 0.000,B 0.000,C 90.000,E1 324.975} C_DIS
LIN {X -0.042,Y -237.967,Z 757.784,A 0.000,B 0.000,C 90.000,E1 321.170} C_DIS
LIN {X -0.104,Y -247.257,Z 757.764,A 0.000,B 0.000,C 90.000,E1 317.472} C_DIS
LIN {X 0.122,Y -257.574,Z 757.743,A 0.000,B 0.000,C 90.000,E1 313.785} C_DIS
LIN {X -0.008,Y -268.796,Z 757.724,A 0.000,B 0.000,C 90.000,E1 310.253} C_DIS
LIN {X -0.099,Y -281.164,Z 757.704,A 0.000,B 0.000,C 90.000,E1 306.790} C_DIS
LIN {X 0.001,Y -293.367,Z 757.687,A 0.000,B 0.000,C 90.000,E1 303.706} C_DIS
LIN {X -0.080,Y -303.974,Z 757.674,A 0.000,B 0.000,C 90.000,E1 301.386} C_DIS
LIN {X 0.068,Y -320.992,Z 757.656,A 0.000,B 0.000,C 90.000,E1 298.103} C_DIS
LIN {X -0.027,Y -333.805,Z 757.644,A 0.000,B 0.000,C 90.000,E1 295.899} C_DIS
LIN {X 0.179,Y -349.470,Z 757.630,A 0.000,B 0.000,C 90.000,E1 293.387} C_DIS
LIN {X -0.124,Y -370.740,Z 757.613,A 0.000,B 0.000,C 90.000,E1 290.429} C_DIS
LIN {X 0.011,Y -396.614,Z 757.596,A 0.000,B 0.000,C 90.000,E1 287.221} C_DIS
LIN {X -0.175,Y -408.888,Z 757.588,A 0.000,B 0.000,C 90.000,E1 285.843} C_DIS
LIN {X 0.092,Y -420.848,Z 757.580,A 0.000,B 0.000,C 90.000,E1 284.426} C_DIS
LIN {X 0.146,Y -432.538,Z 757.573,A 0.000,B 0.000,C 90.000,E1 283.063} C_DIS
LIN {X 0.061,Y -441.700,Z 757.567,A 0.000,B 0.000,C 90.000,E1 282.007} C_DIS
LIN {X 0.081,Y -450.365,Z 757.561,A 0.000,B 0.000,C 90.000,E1 280.950} C_DIS
LIN {X -0.068,Y -460.570,Z 757.554,A 0.000,B 0.000,C 90.000,E1 279.670} C_DIS
LIN {X -0.139,Y -470.319,Z 757.547,A 0.000,B 0.000,C 90.000,E1 278.398} C_DIS
LIN {X 0.132,Y -477.477,Z 757.541,A 0.000,B 0.000,C 90.000,E1 277.352} C_DIS
LIN {X -0.207,Y -480.695,Z 757.538,A 0.000,B 0.000,C 90.000,E1 276.891} C_DIS
LIN {X -0.235,Y -484.831,Z 757.534,A 0.000,B 0.000,C 90.000,E1 276.144} C_DIS
LIN {X -0.050,Y -487.182,Z 757.531,A 0.000,B 0.000,C 90.000,E1 275.625} C_DIS
LIN {X 0.150,Y -489.206,Z 757.528,A 0.000,B 0.000,C 90.000,E1 275.106} C_DIS
LIN {X -0.132,Y -490.840,Z 757.526,A 0.000,B 0.000,C 90.000,E1 274.645} C_DIS
LIN {X 0.046,Y -492.077,Z 757.523,A 0.000,B 0.000,C 90.000,E1 274.131} C_DIS
LIN {X -0.219,Y -492.933,Z 757.520,A 0.000,B 0.000,C 90.000,E1 273.669} C_DIS
LIN {X -0.017,Y -493.389,Z 757.518,A 0.000,B 0.000,C 90.000,E1 273.154} C_DIS
LIN {X 0.217,Y -493.352,Z 757.515,A 0.000,B 0.000,C 90.000,E1 272.636} C_DIS
LIN {X -0.062,Y -492.950,Z 757.512,A 0.000,B 0.000,C 90.000,E1 272.178} C_DIS
LIN {X 0.167,Y -492.096,Z 757.509,A 0.000,B 0.000,C 90.000,E1 271.661} C_DIS
LIN {X -0.114,Y -490.704,Z 757.507,A 0.000,B 0.000,C 90.000,E1 271.203} C_DIS
LIN {X 0.093,Y -488.849,Z 757.504,A 0.000,B 0.000,C 90.000,E1 270.688} C_DIS
LIN {X -0.196,Y -486.431,Z 757.501,A 0.000,B 0.000,C 90.000,E1 270.229} C_DIS
LIN {X -0.013,Y -483.313,Z 757.498,A 0.000,B 0.000,C 90.000,E1 269.714} C_DIS
LIN {X 0.150,Y -479.452,Z 757.496,A 0.000,B 0.000,C 90.000,E1 269.198} C_DIS
LIN {X -0.186,Y -474.719,Z 757.493,A 0.000,B 0.000,C 90.000,E1 268.740} C_DIS
LIN {X 0.114,Y -471.976,Z 757.491,A 0.000,B 0.000,C 90.000,E1 268.453} C_DIS
LIN {X 0.075,Y -466.032,Z 757.489,A 0.000,B 0.000,C 90.000,E1 267.993} C_DIS
LIN {X 0.081,Y -459.610,Z 757.487,A 0.000,B 0.000,C 90.000,E1 267.593} C_DIS
LIN {X 0.124,Y -452.682,Z 757.485,A 0.000,B 0.000,C 90.000,E1 267.249} C_DIS
LIN {X -0.227,Y -445.403,Z 757.483,A 0.000,B 0.000,C 90.000,E1 267.020} C_DIS
LIN {X -0.062,Y -437.370,Z 757.482,A 0.000,B 0.000,C 90.000,E1 266.788} C_DIS
LIN {X 0.107,Y -428.513,Z 757.481,A 0.000,B 0.000,C 90.000,E1 266.617} C_DIS
LIN {X 0.016,Y -420.488,Z 757.481,A 0.000,B 0.000,C 90.000,E1 266.560} C_DIS
LIN {X -0.023,Y -180.953,Z 757.481,A 0.000,B 0.000,C 90.000,E1 266.560} C_DIS
LIN {X -0.085,Y -180.808,Z 757.471,A 0.000,B 0.000,C 90.000,E1 264.837} C_DIS
LIN {X -0.007,Y -178.910,Z 757.443,A 0.000,B 0.000,C 90.000,E1 259.746} C_DIS
LIN {X 0.072,Y -175.953,Z 757.415,A 0.000,B 0.000,C 90.000,E1 254.629} C_DIS
LIN {X 0.019,Y -175.421,Z 757.410,A 0.000,B 0.000,C 90.000,E1 253.795} C_DIS
LIN {X 0.021,Y -172.183,Z 757.386,A 0.000,B 0.000,C 90.000,E1 249.518} C_DIS
LIN {X 0.061,Y -171.655,Z 757.381,A 0.000,B 0.000,C 90.000,E1 248.646} C_DIS
LIN {X 0.055,Y -167.879,Z 757.357,A 0.000,B 0.000,C 90.000,E1 244.332} C_DIS
LIN {X -0.002,Y -166.614,Z 757.348,A 0.000,B 0.000,C 90.000,E1 242.615} C_DIS
LIN {X -0.008,Y -162.602,Z 757.324,A 0.000,B 0.000,C 90.000,E1 238.250} C_DIS
LIN {X -0.034,Y -161.287,Z 757.314,A 0.000,B 0.000,C 90.000,E1 236.501} C_DIS
LIN {X 0.000,Y -157.285,Z 757.289,A 0.000,B 0.000,C 90.000,E1 232.065} C_DIS
LIN {X 0.024,Y -156.004,Z 757.279,A 0.000,B 0.000,C 90.000,E1 230.275} C_DIS
LIN {X -0.017,Y -152.261,Z 757.254,A 0.000,B 0.000,C 90.000,E1 225.810} C_DIS
LIN {X 0.006,Y -150.499,Z 757.239,A 0.000,B 0.000,C 90.000,E1 223.095} C_DIS
LIN {X 0.035,Y -147.224,Z 757.214,A 0.000,B 0.000,C 90.000,E1 218.543} C_DIS
LIN {X 0.005,Y -145.246,Z 757.194,A 0.000,B 0.000,C 90.000,E1 214.898} C_DIS
LIN {X -0.079,Y -142.364,Z 757.163,A 0.000,B 0.000,C 90.000,E1 209.411} C_DIS
LIN {X 0.042,Y -141.750,Z 757.153,A 0.000,B 0.000,C 90.000,E1 207.513} C_DIS
LIN {X -0.032,Y -139.493,Z 757.117,A 0.000,B 0.000,C 90.000,E1 201.046} C_DIS
LIN {X 0.005,Y -138.997,Z 757.101,A 0.000,B 0.000,C 90.000,E1 198.236} C_DIS
LIN {X -0.039,Y -138.337,Z 757.055,A 0.000,B 0.000,C 90.000,E1 189.849} C_DIS
LIN {X -0.016,Y -139.412,Z 757.008,A 0.000,B 0.000,C 90.000,E1 181.432} C_DIS
LIN {X 0.038,Y -141.326,Z 756.972,A 0.000,B 0.000,C 90.000,E1 174.894} C_DIS
LIN {X -0.006,Y -142.684,Z 756.956,A 0.000,B 0.000,C 90.000,E1 172.129} C_DIS
LIN {X -0.025,Y -145.042,Z 756.931,A 0.000,B 0.000,C 90.000,E1 167.521} C_DIS
LIN {X -0.029,Y -147.667,Z 756.910,A 0.000,B 0.000,C 90.000,E1 163.850} C_DIS
LIN {X 0.006,Y -150.310,Z 756.890,A 0.000,B 0.000,C 90.000,E1 160.188} C_DIS
LIN {X 0.018,Y -153.721,Z 756.870,A 0.000,B 0.000,C 90.000,E1 156.561} C_DIS
LIN {X -0.069,Y -157.135,Z 756.850,A 0.000,B 0.000,C 90.000,E1 152.999} C_DIS
LIN {X 0.005,Y -161.281,Z 756.830,A 0.000,B 0.000,C 90.000,E1 149.410} C_DIS
LIN {X 0.023,Y -164.399,Z 756.815,A 0.000,B 0.000,C 90.000,E1 146.755} C_DIS
LIN {X 0.020,Y -169.077,Z 756.796,A 0.000,B 0.000,C 90.000,E1 143.256} C_DIS
LIN {X -0.028,Y -171.636,Z 756.786,A 0.000,B 0.000,C 90.000,E1 141.537} C_DIS
LIN {X 0.018,Y -176.596,Z 756.767,A 0.000,B 0.000,C 90.000,E1 138.081} C_DIS
LIN {X 0.020,Y -180.894,Z 756.753,A 0.000,B 0.000,C 90.000,E1 135.526} C_DIS
LIN {X 0.012,Y -186.309,Z 756.734,A 0.000,B 0.000,C 90.000,E1 132.162} C_DIS
LIN {X -0.056,Y -191.404,Z 756.719,A 0.000,B 0.000,C 90.000,E1 129.402} C_DIS
LIN {X -0.011,Y -192.117,Z 756.716,A 0.000,B 0.000,C 90.000,E1 128.955} C_DIS
LIN {X -0.053,Y -291.508,Z 756.716,A 0.000,B 0.000,C 90.000,E1 128.955} C_DIS
LIN {X 0.057,Y -295.295,Z 756.716,A 0.000,B 0.000,C 90.000,E1 128.830} C_DIS
LIN {X 0.066,Y -298.521,Z 756.715,A 0.000,B 0.000,C 90.000,E1 128.624} C_DIS
LIN {X -0.028,Y -302.169,Z 756.713,A 0.000,B 0.000,C 90.000,E1 128.257} C_DIS
LIN {X 0.064,Y -305.665,Z 756.709,A 0.000,B 0.000,C 90.000,E1 127.649} C_DIS
LIN {X 0.076,Y -307.031,Z 756.707,A 0.000,B 0.000,C 90.000,E1 127.317} C_DIS
LIN {X -0.156,Y -309.952,Z 756.702,A 0.000,B 0.000,C 90.000,E1 126.377} C_DIS
LIN {X 0.140,Y -320.084,Z 756.684,A 0.000,B 0.000,C 90.000,E1 123.086} C_DIS
LIN {X -0.025,Y -330.524,Z 756.668,A 0.000,B 0.000,C 90.000,E1 120.256} C_DIS
LIN {X -0.104,Y -342.321,Z 756.652,A 0.000,B 0.000,C 90.000,E1 117.462} C_DIS
LIN {X 0.001,Y -355.575,Z 756.637,A 0.000,B 0.000,C 90.000,E1 114.695} C_DIS
LIN {X 0.140,Y -368.680,Z 756.624,A 0.000,B 0.000,C 90.000,E1 112.280} C_DIS
LIN {X 0.144,Y -383.126,Z 756.611,A 0.000,B 0.000,C 90.000,E1 109.939} C_DIS
LIN {X -0.135,Y -399.018,Z 756.598,A 0.000,B 0.000,C 90.000,E1 107.692} C_DIS
LIN {X 0.115,Y -416.469,Z 756.586,A 0.000,B 0.000,C 90.000,E1 105.426} C_DIS
LIN {X -0.207,Y -435.585,Z 756.574,A 0.000,B 0.000,C 90.000,E1 103.300} C_DIS
LIN {X -0.014,Y -455.717,Z 756.562,A 0.000,B 0.000,C 90.000,E1 101.243} C_DIS
LIN {X -0.149,Y -468.495,Z 756.556,A 0.000,B 0.000,C 90.000,E1 100.074} C_DIS
LIN {X -0.242,Y -470.464,Z 756.555,A 0.000,B 0.000,C 90.000,E1 99.849} C_DIS
LIN {X 0.211,Y -471.962,Z 756.553,A 0.000,B 0.000,C 90.000,E1 99.557} C_DIS
LIN {X 0.066,Y -473.173,Z 756.552,A 0.000,B 0.000,C 90.000,E1 99.321} C_DIS
LIN {X -0.156,Y -474.058,Z 756.550,A 0.000,B 0.000,C 90.000,E1 99.095} C_DIS
LIN {X 0.036,Y -475.005,Z 756.548,A 0.000,B 0.000,C 90.000,E1 98.568} C_DIS
LIN {X 0.160,Y -474.971,Z 756.545,A 0.000,B 0.000,C 90.000,E1 98.049} C_DIS
LIN {X -0.178,Y -473.956,Z 756.542,A 0.000,B 0.000,C 90.000,E1 97.587} C_DIS
LIN {X 0.152,Y -473.036,Z 756.541,A 0.000,B 0.000,C 90.000,E1 97.296} C_DIS
LIN {X -0.046,Y -471.787,Z 756.539,A 0.000,B 0.000,C 90.000,E1 97.068} C_DIS
LIN {X 0.086,Y -460.296,Z 756.529,A 0.000,B 0.000,C 90.000,E1 95.277} C_DIS
LIN {X 0.025,Y -441.976,Z 756.512,A 0.000,B 0.000,C 90.000,E1 92.178} C_DIS
LIN {X 0.190,Y -432.924,Z 756.503,A 0.000,B 0.000,C 90.000,E1 90.573} C_DIS
LIN {X 0.182,Y -423.486,Z 756.494,A 0.000,B 0.000,C 90.000,E1 88.969} C_DIS
LIN {X 0.112,Y -412.392,Z 756.484,A 0.000,B 0.000,C 90.000,E1 87.078} C_DIS
LIN {X -0.133,Y -401.142,Z 756.473,A 0.000,B 0.000,C 90.000,E1 85.179} C_DIS
LIN {X -0.143,Y -388.253,Z 756.461,A 0.000,B 0.000,C 90.000,E1 82.932} C_DIS
LIN {X -0.019,Y -372.685,Z 756.445,A 0.000,B 0.000,C 90.000,E1 80.038} C_DIS
LIN {X 0.135,Y -356.398,Z 756.427,A 0.000,B 0.000,C 90.000,E1 76.769} C_DIS
LIN {X -0.179,Y -343.516,Z 756.411,A 0.000,B 0.000,C 90.000,E1 74.102} C_DIS
LIN {X -0.163,Y -333.754,Z 756.400,A 0.000,B 0.000,C 90.000,E1 71.945} C_DIS
LIN {X 0.020,Y -320.299,Z 756.382,A 0.000,B 0.000,C 90.000,E1 68.773} C_DIS
LIN {X 0.049,Y -306.567,Z 756.362,A 0.000,B 0.000,C 90.000,E1 65.229} C_DIS
LIN {X -0.131,Y -294.321,Z 756.342,A 0.000,B 0.000,C 90.000,E1 61.641} C_DIS
LIN {X 0.050,Y -284.131,Z 756.324,A 0.000,B 0.000,C 90.000,E1 58.250} C_DIS
LIN {X 0.072,Y -276.405,Z 756.308,A 0.000,B 0.000,C 90.000,E1 55.515} C_DIS
LIN {X -0.014,Y -268.869,Z 756.293,A 0.000,B 0.000,C 90.000,E1 52.763} C_DIS
LIN {X 0.068,Y -263.205,Z 756.281,A 0.000,B 0.000,C 90.000,E1 50.642} C_DIS
LIN {X 0.093,Y -255.565,Z 756.266,A 0.000,B 0.000,C 90.000,E1 47.796} C_DIS
LIN {X 0.042,Y -249.835,Z 756.254,A 0.000,B 0.000,C 90.000,E1 45.648} C_DIS
LIN {X -0.122,Y -242.231,Z 756.237,A 0.000,B 0.000,C 90.000,E1 42.771} C_DIS
LIN {X -0.101,Y -234.621,Z 756.221,A 0.000,B 0.000,C 90.000,E1 39.806} C_DIS
LIN {X 0.019,Y -225.601,Z 756.200,A 0.000,B 0.000,C 90.000,E1 36.011} C_DIS
LIN {X -0.122,Y -217.241,Z 756.179,A 0.000,B 0.000,C 90.000,E1 32.212} C_DIS
LIN {X -0.052,Y -211.251,Z 756.161,A 0.000,B 0.000,C 90.000,E1 29.077} C_DIS
LIN {X 0.026,Y -206.018,Z 756.144,A 0.000,B 0.000,C 90.000,E1 25.899} C_DIS
LIN {X 0.051,Y -200.447,Z 756.122,A 0.000,B 0.000,C 90.000,E1 21.897} C_DIS
LIN {X -0.012,Y -195.984,Z 756.099,A 0.000,B 0.000,C 90.000,E1 17.873} C_DIS
LIN {X 0.062,Y -192.088,Z 756.072,A 0.000,B 0.000,C 90.000,E1 12.952} C_DIS
LIN {X 0.079,Y -189.353,Z 756.040,A 0.000,B 0.000,C 90.000,E1 7.182} C_DIS
LIN {X -0.004,Y -190.617,Z 755.965,A 0.000,B 0.000,C 90.000,E1 353.742} C_DIS
LIN {X -0.041,Y -193.672,Z 755.938,A 0.000,B 0.000,C 90.000,E1 348.814} C_DIS
LIN {X 0.048,Y -197.390,Z 755.915,A 0.000,B 0.000,C 90.000,E1 344.700} C_DIS
LIN {X -0.061,Y -202.058,Z 755.893,A 0.000,B 0.000,C 90.000,E1 340.678} C_DIS
LIN {X -0.055,Y -207.736,Z 755.870,A 0.000,B 0.000,C 90.000,E1 336.666} C_DIS
LIN {X -0.002,Y -214.217,Z 755.848,A 0.000,B 0.000,C 90.000,E1 332.692} C_DIS
LIN {X -0.007,Y -221.560,Z 755.827,A 0.000,B 0.000,C 90.000,E1 328.791} C_DIS
LIN {X -0.045,Y -227.843,Z 755.810,A 0.000,B 0.000,C 90.000,E1 325.722} C_DIS
LIN {X -0.045,Y -234.490,Z 755.793,A 0.000,B 0.000,C 90.000,E1 322.683} C_DIS
LIN {X 0.041,Y -241.599,Z 755.776,A 0.000,B 0.000,C 90.000,E1 319.666} C_DIS
LIN {X 0.082,Y -251.303,Z 755.755,A 0.000,B 0.000,C 90.000,E1 315.972} C_DIS
LIN {X 0.090,Y -261.966,Z 755.735,A 0.000,B 0.000,C 90.000,E1 312.366} C_DIS
LIN {X 0.128,Y -273.612,Z 755.716,A 0.000,B 0.000,C 90.000,E1 308.830} C_DIS
LIN {X 0.079,Y -286.407,Z 755.697,A 0.000,B 0.000,C 90.000,E1 305.391} C_DIS
LIN {X 0.182,Y -299.284,Z 755.680,A 0.000,B 0.000,C 90.000,E1 302.339} C_DIS
LIN {X 0.042,Y -308.902,Z 755.669,A 0.000,B 0.000,C 90.000,E1 300.384} C_DIS
LIN {X -0.083,Y -326.422,Z 755.651,A 0.000,B 0.000,C 90.000,E1 297.180} C_DIS
LIN {X 0.062,Y -345.355,Z 755.634,A 0.000,B 0.000,C 90.000,E1 294.027} C_DIS
LIN {X -0.101,Y -366.242,Z 755.617,A 0.000,B 0.000,C 90.000,E1 291.025} C_DIS
LIN {X 0.211,Y -389.180,Z 755.600,A 0.000,B 0.000,C 90.000,E1 288.055} C_DIS
LIN {X -0.045,Y -406.048,Z 755.590,A 0.000,B 0.000,C 90.000,E1 286.134} C_DIS
LIN {X 0.183,Y -418.048,Z 755.582,A 0.000,B 0.000,C 90.000,E1 284.717} C_DIS
LIN {X 0.189,Y -429.800,Z 755.574,A 0.000,B 0.000,C 90.000,E1 283.355} C_DIS
LIN {X -0.059,Y -441.128,Z 755.567,A 0.000,B 0.000,C 90.000,E1 282.063} C_DIS
LIN {X -0.051,Y -449.809,Z 755.561,A 0.000,B 0.000,C 90.000,E1 281.007} C_DIS
LIN {X 0.241,Y -460.041,Z 755.554,A 0.000,B 0.000,C 90.000,E1 279.670} C_DIS
LIN {X 0.169,Y -469.828,Z 755.547,A 0.000,B 0.000,C 90.000,E1 278.398} C_DIS
LIN {X -0.034,Y -477.059,Z 755.541,A 0.000,B 0.000,C 90.000,E1 277.409} C_DIS
LIN {X -0.095,Y -481.780,Z 755.537,A 0.000,B 0.000,C 90.000,E1 276.663} C_DIS
LIN {X -0.053,Y -485.783,Z 755.533,A 0.000,B 0.000,C 90.000,E1 275.910} C_DIS
LIN {X -0.032,Y -489.001,Z 755.529,A 0.000,B 0.000,C 90.000,E1 275.163} C_DIS
LIN {X 0.178,Y -490.690,Z 755.526,A 0.000,B 0.000,C 90.000,E1 274.645} C_DIS
LIN {X -0.134,Y -491.996,Z 755.523,A 0.000,B 0.000,C 90.000,E1 274.188} C_DIS
LIN {X 0.091,Y -492.885,Z 755.520,A 0.000,B 0.000,C 90.000,E1 273.669} C_DIS
LIN {X -0.200,Y -493.365,Z 755.518,A 0.000,B 0.000,C 90.000,E1 273.212} C_DIS
LIN {X 0.034,Y -493.388,Z 755.515,A 0.000,B 0.000,C 90.000,E1 272.694} C_DIS
LIN {X -0.245,Y -493.011,Z 755.512,A 0.000,B 0.000,C 90.000,E1 272.236} C_DIS
LIN {X -0.015,Y -492.216,Z 755.510,A 0.000,B 0.000,C 90.000,E1 271.718} C_DIS
LIN {X 0.195,Y -490.905,Z 755.507,A 0.000,B 0.000,C 90.000,E1 271.203} C_DIS
LIN {X -0.088,Y -489.090,Z 755.504,A 0.000,B 0.000,C 90.000,E1 270.745} C_DIS
LIN {X 0.112,Y -486.742,Z 755.501,A 0.000,B 0.000,C 90.000,E1 270.229} C_DIS
LIN {X -0.189,Y -483.720,Z 755.499,A 0.000,B 0.000,C 90.000,E1 269.771} C_DIS
LIN {X -0.022,Y -479.929,Z 755.496,A 0.000,B 0.000,C 90.000,E1 269.255} C_DIS
LIN {X 0.122,Y -475.296,Z 755.493,A 0.000,B 0.000,C 90.000,E1 268.740} C_DIS
LIN {X -0.050,Y -472.628,Z 755.492,A 0.000,B 0.000,C 90.000,E1 268.511} C_DIS
LIN {X -0.119,Y -466.736,Z 755.489,A 0.000,B 0.000,C 90.000,E1 268.051} C_DIS
LIN {X -0.035,Y -463.509,Z 755.488,A 0.000,B 0.000,C 90.000,E1 267.822} C_DIS
LIN {X 0.132,Y -456.768,Z 755.486,A 0.000,B 0.000,C 90.000,E1 267.421} C_DIS
LIN {X -0.099,Y -449.433,Z 755.484,A 0.000,B 0.000,C 90.000,E1 267.135} C_DIS
LIN {X 0.200,Y -441.849,Z 755.483,A 0.000,B 0.000,C 90.000,E1 266.849} C_DIS
LIN {X 0.098,Y -433.061,Z 755.482,A 0.000,B 0.000,C 90.000,E1 266.674} C_DIS
LIN {X 0.039,Y -423.123,Z 755.481,A 0.000,B 0.000,C 90.000,E1 266.560} C_DIS
LIN {X -0.104,Y -418.511,Z 755.481,A 0.000,B 0.000,C 90.000,E1 266.560} C_DIS
LIN {X -0.076,Y -180.951,Z 755.481,A 0.000,B 0.000,C 90.000,E1 266.560} C_DIS
LIN {X 0.068,Y -180.805,Z 755.471,A 0.000,B 0.000,C 90.000,E1 264.780} C_DIS
LIN {X -0.035,Y -178.906,Z 755.443,A 0.000,B 0.000,C 90.000,E1 259.746} C_DIS
LIN {X 0.045,Y -175.950,Z 755.415,A 0.000,B 0.000,C 90.000,E1 254.629} C_DIS
LIN {X -0.008,Y -175.414,Z 755.410,A 0.000,B 0.000,C 90.000,E1 253.795} C_DIS
LIN {X -0.005,Y -172.178,Z 755.386,A 0.000,B 0.000,C 90.000,E1 249.518} C_DIS
LIN {X 0.034,Y -171.648,Z 755.381,A 0.000,B 0.000,C 90.000,E1 248.646} C_DIS
LIN {X 0.028,Y -167.872,Z 755.357,A 0.000,B 0.000,C 90.000,E1 244.332} C_DIS
LIN {X -0.029,Y -166.607,Z 755.348,A 0.000,B 0.000,C 90.000,E1 242.615} C_DIS
LIN {X -0.034,Y -162.595,Z 755.324,A 0.000,B 0.000,C 90.000,E1 238.250} C_DIS
LIN {X -0.060,Y -161.279,Z 755.314,A 0.000,B 0.000,C 90.000,E1 236.501} C_DIS
LIN {X -0.025,Y -157.278,Z 755.289,A 0.000,B 0.000,C 90.000,E1 232.065} C_DIS
LIN {X -0.001,Y -155.997,Z 755.279,A 0.000,B 0.000,C 90.000,E1 230.275} C_DIS
LIN {X -0.042,Y -152.255,Z 755.254,A 0.000,B 0.000,C 90.000,E1 225.810} C_DIS
LIN {X -0.019,Y -150.494,Z 755.239,A 0.000,B 0.000,C 90.000,E1 223.095} C_DIS
LIN {X 0.011,Y -147.217,Z 755.214,A 0.000,B 0.000,C 90.000,E1 218.543} C_DIS
LIN {X -0.019,Y -145.240,Z 755.194,A 0.000,B 0.000,C 90.000,E1 214.898} C_DIS
LIN {X 0.021,Y -142.360,Z 755.163,A 0.000,B 0.000,C 90.000,E1 209.361} C_DIS
LIN {X 0.019,Y -141.747,Z 755.153,A 0.000,B 0.000,C 90.000,E1 207.513} C_DIS
LIN {X -0.055,Y -139.491,Z 755.117,A 0.000,B 0.000,C 90.000,E1 201.046} C_DIS
LIN {X -0.018,Y -138.995,Z 755.101,A 0.000,B 0.000,C 90.000,E1 198.236} C_DIS
LIN {X -0.062,Y -138.336,Z 755.055,A 0.000,B 0.000,C 90.000,E1 189.849} C_DIS
LIN {X -0.040,Y -139.415,Z 755.008,A 0.000,B 0.000,C 90.000,E1 181.432} C_DIS
LIN {X 0.014,Y -141.330,Z 754.972,A 0.000,B 0.000,C 90.000,E1 174.894} C_DIS
LIN {X -0.029,Y -142.687,Z 754.956,A 0.000,B 0.000,C 90.000,E1 172.129} C_DIS
LIN {X -0.050,Y -145.048,Z 754.931,A 0.000,B 0.000,C 90.000,E1 167.521} C_DIS
LIN {X -0.053,Y -147.673,Z 754.910,A 0.000,B 0.000,C 90.000,E1 163.850} C_DIS
LIN {X -0.018,Y -150.317,Z 754.890,A 0.000,B 0.000,C 90.000,E1 160.188} C_DIS
LIN {X 0.054,Y -153.730,Z 754.870,A 0.000,B 0.000,C 90.000,E1 156.538} C_DIS
LIN {X 0.045,Y -157.145,Z 754.850,A 0.000,B 0.000,C 90.000,E1 152.948} C_DIS
LIN {X -0.020,Y -161.293,Z 754.830,A 0.000,B 0.000,C 90.000,E1 149.410} C_DIS
LIN {X -0.002,Y -164.409,Z 754.815,A 0.000,B 0.000,C 90.000,E1 146.755} C_DIS
LIN {X -0.006,Y -169.091,Z 754.796,A 0.000,B 0.000,C 90.000,E1 143.256} C_DIS
LIN {X -0.055,Y -171.647,Z 754.786,A 0.000,B 0.000,C 90.000,E1 141.537} C_DIS
LIN {X -0.008,Y -176.610,Z 754.767,A 0.000,B 0.000,C 90.000,E1 138.081} C_DIS
LIN {X -0.007,Y -180.908,Z 754.753,A 0.000,B 0.000,C 90.000,E1 135.526} C_DIS
LIN {X -0.017,Y -186.325,Z 754.734,A 0.000,B 0.000,C 90.000,E1 132.162} C_DIS
LIN {X 0.065,Y -191.417,Z 754.719,A 0.000,B 0.000,C 90.000,E1 129.358} C_DIS
LIN {X 0.034,Y -192.094,Z 754.716,A 0.000,B 0.000,C 90.000,E1 128.955} C_DIS
LIN {X 0.017,Y -291.534,Z 754.716,A 0.000,B 0.000,C 90.000,E1 128.955} C_DIS
LIN {X 0.014,Y -295.706,Z 754.716,A 0.000,B 0.000,C 90.000,E1 128.830} C_DIS
LIN {X 0.003,Y -298.777,Z 754.715,A 0.000,B 0.000,C 90.000,E1 128.624} C_DIS
LIN {X -0.029,Y -302.475,Z 754.712,A 0.000,B 0.000,C 90.000,E1 128.222} C_DIS
LIN {X 0.108,Y -304.407,Z 754.711,A 0.000,B 0.000,C 90.000,E1 127.890} C_DIS
LIN {X 0.007,Y -305.925,Z 754.709,A 0.000,B 0.000,C 90.000,E1 127.604} C_DIS
LIN {X -0.031,Y -307.218,Z 754.707,A 0.000,B 0.000,C 90.000,E1 127.282} C_DIS
LIN {X 0.044,Y -319.158,Z 754.685,A 0.000,B 0.000,C 90.000,E1 123.372} C_DIS
LIN {X -0.147,Y -329.477,Z 754.670,A 0.000,B 0.000,C 90.000,E1 120.541} C_DIS
LIN {X -0.088,Y -341.141,Z 754.654,A 0.000,B 0.000,C 90.000,E1 117.719} C_DIS
LIN {X -0.021,Y -354.259,Z 754.639,A 0.000,B 0.000,C 90.000,E1 114.951} C_DIS
LIN {X 0.226,Y -367.229,Z 754.625,A 0.000,B 0.000,C 90.000,E1 112.514} C_DIS
LIN {X 0.056,Y -381.531,Z 754.612,A 0.000,B 0.000,C 90.000,E1 110.194} C_DIS
LIN {X 0.244,Y -397.266,Z 754.599,A 0.000,B 0.000,C 90.000,E1 107.873} C_DIS
LIN {X 0.067,Y -414.549,Z 754.587,A 0.000,B 0.000,C 90.000,E1 105.662} C_DIS
LIN {X 0.098,Y -433.508,Z 754.575,A 0.000,B 0.000,C 90.000,E1 103.480} C_DIS
LIN {X 0.163,Y -453.579,Z 754.564,A 0.000,B 0.000,C 90.000,E1 101.422} C_DIS
LIN {X -0.002,Y -468.833,Z 754.556,A 0.000,B 0.000,C 90.000,E1 100.018} C_DIS
LIN {X -0.125,Y -470.747,Z 754.554,A 0.000,B 0.000,C 90.000,E1 99.792} C_DIS
LIN {X -0.166,Y -472.201,Z 754.553,A 0.000,B 0.000,C 90.000,E1 99.557} C_DIS
LIN {X 0.011,Y -474.190,Z 754.550,A 0.000,B 0.000,C 90.000,E1 99.029} C_DIS
LIN {X 0.122,Y -475.053,Z 754.547,A 0.000,B 0.000,C 90.000,E1 98.511} C_DIS
LIN {X -0.221,Y -474.938,Z 754.545,A 0.000,B 0.000,C 90.000,E1 98.049} C_DIS
LIN {X -0.090,Y -473.836,Z 754.542,A 0.000,B 0.000,C 90.000,E1 97.530} C_DIS
LIN {X -0.228,Y -472.864,Z 754.540,A 0.000,B 0.000,C 90.000,E1 97.296} C_DIS
LIN {X 0.101,Y -471.552,Z 754.539,A 0.000,B 0.000,C 90.000,E1 97.004} C_DIS
LIN {X 0.014,Y -452.214,Z 754.522,A 0.000,B 0.000,C 90.000,E1 93.955} C_DIS
LIN {X -0.156,Y -440.255,Z 754.510,A 0.000,B 0.000,C 90.000,E1 91.892} C_DIS
LIN {X -0.175,Y -432.679,Z 754.503,A 0.000,B 0.000,C 90.000,E1 90.573} C_DIS
LIN {X -0.179,Y -423.251,Z 754.494,A 0.000,B 0.000,C 90.000,E1 88.969} C_DIS
LIN {X 0.168,Y -412.175,Z 754.484,A 0.000,B 0.000,C 90.000,E1 87.020} C_DIS
LIN {X -0.084,Y -400.925,Z 754.473,A 0.000,B 0.000,C 90.000,E1 85.122} C_DIS
LIN {X -0.101,Y -388.072,Z 754.460,A 0.000,B 0.000,C 90.000,E1 82.875} C_DIS
LIN {X 0.013,Y -372.515,Z 754.444,A 0.000,B 0.000,C 90.000,E1 79.982} C_DIS
LIN {X -0.109,Y -356.253,Z 754.426,A 0.000,B 0.000,C 90.000,E1 76.756} C_DIS
LIN {X -0.072,Y -343.384,Z 754.411,A 0.000,B 0.000,C 90.000,E1 74.031} C_DIS
LIN {X -0.177,Y -332.244,Z 754.398,A 0.000,B 0.000,C 90.000,E1 71.583} C_DIS
LIN {X -0.096,Y -317.620,Z 754.378,A 0.000,B 0.000,C 90.000,E1 68.103} C_DIS
LIN {X -0.032,Y -304.221,Z 754.359,A 0.000,B 0.000,C 90.000,E1 64.537} C_DIS
LIN {X -0.138,Y -292.318,Z 754.338,A 0.000,B 0.000,C 90.000,E1 60.923} C_DIS
LIN {X -0.024,Y -282.324,Z 754.320,A 0.000,B 0.000,C 90.000,E1 57.533} C_DIS
LIN {X 0.099,Y -274.673,Z 754.304,A 0.000,B 0.000,C 90.000,E1 54.769} C_DIS
LIN {X 0.123,Y -267.183,Z 754.289,A 0.000,B 0.000,C 90.000,E1 51.984} C_DIS
LIN {X -0.036,Y -261.531,Z 754.277,A 0.000,B 0.000,C 90.000,E1 49.908} C_DIS
LIN {X 0.044,Y -255.806,Z 754.265,A 0.000,B 0.000,C 90.000,E1 47.757} C_DIS
LIN {X 0.011,Y -250.091,Z 754.253,A 0.000,B 0.000,C 90.000,E1 45.607} C_DIS
LIN {X 0.022,Y -242.474,Z 754.237,A 0.000,B 0.000,C 90.000,E1 42.690} C_DIS
LIN {X 0.045,Y -234.845,Z 754.221,A 0.000,B 0.000,C 90.000,E1 39.725} C_DIS
LIN {X 0.030,Y -225.796,Z 754.200,A 0.000,B 0.000,C 90.000,E1 35.964} C_DIS
LIN {X 0.018,Y -217.437,Z 754.179,A 0.000,B 0.000,C 90.000,E1 32.133} C_DIS
LIN {X -0.018,Y -211.413,Z 754.161,A 0.000,B 0.000,C 90.000,E1 29.027} C_DIS
LIN {X 0.069,Y -206.191,Z 754.144,A 0.000,B 0.000,C 90.000,E1 25.848} C_DIS
LIN {X -0.083,Y -200.606,Z 754.122,A 0.000,B 0.000,C 90.000,E1 21.897} C_DIS
LIN {X 0.048,Y -196.117,Z 754.099,A 0.000,B 0.000,C 90.000,E1 17.819} C_DIS
LIN {X -0.014,Y -192.212,Z 754.072,A 0.000,B 0.000,C 90.000,E1 12.939} C_DIS
LIN {X -0.033,Y -189.480,Z 754.040,A 0.000,B 0.000,C 90.000,E1 7.182} C_DIS
LIN {X 0.001,Y -190.716,Z 753.965,A 0.000,B 0.000,C 90.000,E1 353.742} C_DIS
LIN {X -0.033,Y -193.777,Z 753.938,A 0.000,B 0.000,C 90.000,E1 348.814} C_DIS
LIN {X 0.059,Y -197.491,Z 753.915,A 0.000,B 0.000,C 90.000,E1 344.700} C_DIS
LIN {X -0.045,Y -202.147,Z 753.893,A 0.000,B 0.000,C 90.000,E1 340.678} C_DIS
LIN {X -0.037,Y -207.817,Z 753.870,A 0.000,B 0.000,C 90.000,E1 336.666} C_DIS
LIN {X 0.020,Y -214.304,Z 753.848,A 0.000,B 0.000,C 90.000,E1 332.692} C_DIS
LIN {X 0.019,Y -221.635,Z 753.827,A 0.000,B 0.000,C 90.000,E1 328.791} C_DIS
LIN {X -0.017,Y -227.914,Z 753.810,A 0.000,B 0.000,C 90.000,E1 325.722} C_DIS
LIN {X 0.093,Y -236.317,Z 753.788,A 0.000,B 0.000,C 90.000,E1 321.904} C_DIS
LIN {X 0.169,Y -245.399,Z 753.768,A 0.000,B 0.000,C 90.000,E1 318.162} C_DIS
LIN {X -0.039,Y -254.439,Z 753.750,A 0.000,B 0.000,C 90.000,E1 314.919} C_DIS
LIN {X 0.082,Y -265.344,Z 753.730,A 0.000,B 0.000,C 90.000,E1 311.310} C_DIS
LIN {X 0.059,Y -277.343,Z 753.710,A 0.000,B 0.000,C 90.000,E1 307.810} C_DIS
LIN {X -0.017,Y -289.141,Z 753.693,A 0.000,B 0.000,C 90.000,E1 304.739} C_DIS
LIN {X -0.024,Y -300.833,Z 753.678,A 0.000,B 0.000,C 90.000,E1 302.054} C_DIS
LIN {X 0.058,Y -313.961,Z 753.663,A 0.000,B 0.000,C 90.000,E1 299.411} C_DIS
LIN {X -0.047,Y -331.880,Z 753.646,A 0.000,B 0.000,C 90.000,E1 296.232} C_DIS
LIN {X -0.204,Y -347.333,Z 753.632,A 0.000,B 0.000,C 90.000,E1 293.770} C_DIS
LIN {X -0.114,Y -368.318,Z 753.615,A 0.000,B 0.000,C 90.000,E1 290.737} C_DIS
LIN {X -0.091,Y -391.449,Z 753.599,A 0.000,B 0.000,C 90.000,E1 287.819} C_DIS
LIN {X 0.224,Y -406.076,Z 753.589,A 0.000,B 0.000,C 90.000,E1 286.079} C_DIS
LIN {X 0.058,Y -418.037,Z 753.582,A 0.000,B 0.000,C 90.000,E1 284.717} C_DIS
LIN {X -0.187,Y -432.071,Z 753.573,A 0.000,B 0.000,C 90.000,E1 283.119} C_DIS
LIN {X -0.080,Y -443.374,Z 753.565,A 0.000,B 0.000,C 90.000,E1 281.771} C_DIS
LIN {X -0.046,Y -451.892,Z 753.560,A 0.000,B 0.000,C 90.000,E1 280.715} C_DIS
LIN {X -0.172,Y -462.025,Z 753.552,A 0.000,B 0.000,C 90.000,E1 279.434} C_DIS
LIN {X -0.072,Y -469.852,Z 753.547,A 0.000,B 0.000,C 90.000,E1 278.398} C_DIS
LIN {X 0.195,Y -477.099,Z 753.541,A 0.000,B 0.000,C 90.000,E1 277.352} C_DIS
LIN {X 0.138,Y -481.815,Z 753.537,A 0.000,B 0.000,C 90.000,E1 276.606} C_DIS
LIN {X 0.182,Y -485.806,Z 753.533,A 0.000,B 0.000,C 90.000,E1 275.853} C_DIS
LIN {X 0.206,Y -489.029,Z 753.529,A 0.000,B 0.000,C 90.000,E1 275.106} C_DIS
LIN {X -0.072,Y -490.716,Z 753.526,A 0.000,B 0.000,C 90.000,E1 274.645} C_DIS
LIN {X 0.107,Y -492.014,Z 753.523,A 0.000,B 0.000,C 90.000,E1 274.131} C_DIS
LIN {X -0.160,Y -492.890,Z 753.520,A 0.000,B 0.000,C 90.000,E1 273.669} C_DIS
LIN {X 0.043,Y -493.345,Z 753.518,A 0.000,B 0.000,C 90.000,E1 273.154} C_DIS
LIN {X -0.216,Y -493.385,Z 753.515,A 0.000,B 0.000,C 90.000,E1 272.694} C_DIS
LIN {X -0.004,Y -492.961,Z 753.512,A 0.000,B 0.000,C 90.000,E1 272.178} C_DIS
LIN {X 0.226,Y -492.173,Z 753.509,A 0.000,B 0.000,C 90.000,E1 271.661} C_DIS
LIN {X -0.054,Y -490.883,Z 753.507,A 0.000,B 0.000,C 90.000,E1 271.203} C_DIS
LIN {X 0.153,Y -489.073,Z 753.504,A 0.000,B 0.000,C 90.000,E1 270.688} C_DIS
LIN {X -0.136,Y -486.690,Z 753.501,A 0.000,B 0.000,C 90.000,E1 270.229} C_DIS
LIN {X 0.047,Y -483.666,Z 753.498,A 0.000,B 0.000,C 90.000,E1 269.714} C_DIS
LIN {X 0.212,Y -479.866,Z 753.496,A 0.000,B 0.000,C 90.000,E1 269.198} C_DIS
LIN {X -0.121,Y -475.196,Z 753.493,A 0.000,B 0.000,C 90.000,E1 268.740} C_DIS
LIN {X 0.032,Y -469.529,Z 753.490,A 0.000,B 0.000,C 90.000,E1 268.224} C_DIS
LIN {X 0.113,Y -466.592,Z 753.489,A 0.000,B 0.000,C 90.000,E1 267.993} C_DIS
LIN {X 0.062,Y -460.078,Z 753.487,A 0.000,B 0.000,C 90.000,E1 267.593} C_DIS
LIN {X 0.081,Y -453.254,Z 753.485,A 0.000,B 0.000,C 90.000,E1 267.249} C_DIS
LIN {X 0.168,Y -445.828,Z 753.483,A 0.000,B 0.000,C 90.000,E1 266.963} C_DIS
LIN {X 0.123,Y -441.899,Z 753.483,A 0.000,B 0.000,C 90.000,E1 266.849} C_DIS
LIN {X 0.006,Y -433.138,Z 753.482,A 0.000,B 0.000,C 90.000,E1 266.674} C_DIS
LIN {X 0.148,Y -425.937,Z 753.481,A 0.000,B 0.000,C 90.000,E1 266.560} C_DIS
LIN {X -0.147,Y -419.807,Z 753.481,A 0.000,B 0.000,C 90.000,E1 266.560} C_DIS
LIN {X 0.092,Y -180.950,Z 753.481,A 0.000,B 0.000,C 90.000,E1 266.502} C_DIS
LIN {X 0.056,Y -180.804,Z 753.471,A 0.000,B 0.000,C 90.000,E1 264.780} C_DIS
LIN {X -0.046,Y -178.904,Z 753.443,A 0.000,B 0.000,C 90.000,E1 259.746} C_DIS
LIN {X 0.034,Y -175.949,Z 753.415,A 0.000,B 0.000,C 90.000,E1 254.629} C_DIS
LIN {X -0.019,Y -175.411,Z 753.410,A 0.000,B 0.000,C 90.000,E1 253.795} C_DIS
LIN {X -0.016,Y -172.175,Z 753.386,A 0.000,B 0.000,C 90.000,E1 249.518} C_DIS
LIN {X 0.023,Y -171.646,Z 753.381,A 0.000,B 0.000,C 90.000,E1 248.646} C_DIS
LIN {X 0.018,Y -167.869,Z 753.357,A 0.000,B 0.000,C 90.000,E1 244.332} C_DIS
LIN {X -0.039,Y -166.603,Z 753.348,A 0.000,B 0.000,C 90.000,E1 242.615} C_DIS
LIN {X -0.045,Y -162.592,Z 753.324,A 0.000,B 0.000,C 90.000,E1 238.250} C_DIS
LIN {X -0.070,Y -161.275,Z 753.314,A 0.000,B 0.000,C 90.000,E1 236.501} C_DIS
LIN {X -0.035,Y -157.276,Z 753.289,A 0.000,B 0.000,C 90.000,E1 232.065} C_DIS
LIN {X -0.012,Y -155.995,Z 753.279,A 0.000,B 0.000,C 90.000,E1 230.275} C_DIS
LIN {X -0.052,Y -152.252,Z 753.254,A 0.000,B 0.000,C 90.000,E1 225.810} C_DIS
LIN {X -0.029,Y -150.491,Z 753.239,A 0.000,B 0.000,C 90.000,E1 223.095} C_DIS
LIN {X 0.001,Y -147.216,Z 753.214,A 0.000,B 0.000,C 90.000,E1 218.543} C_DIS
LIN {X -0.029,Y -145.237,Z 753.194,A 0.000,B 0.000,C 90.000,E1 214.898} C_DIS
LIN {X 0.081,Y -142.359,Z 753.163,A 0.000,B 0.000,C 90.000,E1 209.333} C_DIS
LIN {X 0.008,Y -141.746,Z 753.153,A 0.000,B 0.000,C 90.000,E1 207.513} C_DIS
LIN {X -0.065,Y -139.490,Z 753.117,A 0.000,B 0.000,C 90.000,E1 201.046} C_DIS
LIN {X -0.028,Y -138.994,Z 753.101,A 0.000,B 0.000,C 90.000,E1 198.236} C_DIS
LIN {X -0.071,Y -138.337,Z 753.055,A 0.000,B 0.000,C 90.000,E1 189.849} C_DIS
LIN {X -0.049,Y -139.416,Z 753.008,A 0.000,B 0.000,C 90.000,E1 181.432} C_DIS
LIN {X 0.004,Y -141.332,Z 752.972,A 0.000,B 0.000,C 90.000,E1 174.894} C_DIS
LIN {X -0.039,Y -142.689,Z 752.956,A 0.000,B 0.000,C 90.000,E1 172.129} C_DIS
LIN {X -0.059,Y -145.051,Z 752.931,A 0.000,B 0.000,C 90.000,E1 167.521} C_DIS
LIN {X 0.079,Y -147.676,Z 752.910,A 0.000,B 0.000,C 90.000,E1 163.795} C_DIS
LIN {X -0.028,Y -150.320,Z 752.890,A 0.000,B 0.000,C 90.000,E1 160.188} C_DIS
LIN {X 0.044,Y -153.735,Z 752.870,A 0.000,B 0.000,C 90.000,E1 156.538} C_DIS
LIN {X 0.035,Y -157.148,Z 752.850,A 0.000,B 0.000,C 90.000,E1 152.948} C_DIS
LIN {X -0.031,Y -161.298,Z 752.830,A 0.000,B 0.000,C 90.000,E1 149.410} C_DIS
LIN {X -0.013,Y -164.414,Z 752.815,A 0.000,B 0.000,C 90.000,E1 146.755} C_DIS
LIN {X -0.017,Y -169.096,Z 752.796,A 0.000,B 0.000,C 90.000,E1 143.256} C_DIS
LIN {X -0.066,Y -171.652,Z 752.786,A 0.000,B 0.000,C 90.000,E1 141.537} C_DIS
LIN {X -0.021,Y -176.616,Z 752.767,A 0.000,B 0.000,C 90.000,E1 138.081} C_DIS
LIN {X 0.108,Y -180.914,Z 752.753,A 0.000,B 0.000,C 90.000,E1 135.486} C_DIS
LIN {X -0.028,Y -186.331,Z 752.734,A 0.000,B 0.000,C 90.000,E1 132.162} C_DIS
LIN {X 0.055,Y -191.421,Z 752.719,A 0.000,B 0.000,C 90.000,E1 129.358} C_DIS
LIN {X -0.025,Y -192.064,Z 752.717,A 0.000,B 0.000,C 90.000,E1 128.991} C_DIS
LIN {X -0.074,Y -291.166,Z 752.717,A 0.000,B 0.000,C 90.000,E1 128.991} C_DIS
LIN {X -0.005,Y -296.004,Z 752.716,A 0.000,B 0.000,C 90.000,E1 128.830} C_DIS
LIN {X 0.056,Y -298.776,Z 752.715,A 0.000,B 0.000,C 90.000,E1 128.624} C_DIS
LIN {X -0.041,Y -302.539,Z 752.712,A 0.000,B 0.000,C 90.000,E1 128.222} C_DIS
LIN {X 0.081,Y -304.457,Z 752.711,A 0.000,B 0.000,C 90.000,E1 127.890} C_DIS
LIN {X -0.036,Y -305.964,Z 752.709,A 0.000,B 0.000,C 90.000,E1 127.604} C_DIS
LIN {X -0.074,Y -307.236,Z 752.707,A 0.000,B 0.000,C 90.000,E1 127.282} C_DIS
LIN {X 0.000,Y -319.163,Z 752.685,A 0.000,B 0.000,C 90.000,E1 123.372} C_DIS
LIN {X -0.025,Y -329.487,Z 752.669,A 0.000,B 0.000,C 90.000,E1 120.512} C_DIS
LIN {X -0.135,Y -341.154,Z 752.654,A 0.000,B 0.000,C 90.000,E1 117.719} C_DIS
LIN {X -0.069,Y -354.275,Z 752.639,A 0.000,B 0.000,C 90.000,E1 114.951} C_DIS
LIN {X 0.177,Y -367.249,Z 752.625,A 0.000,B 0.000,C 90.000,E1 112.514} C_DIS
LIN {X 0.137,Y -381.555,Z 752.612,A 0.000,B 0.000,C 90.000,E1 110.174} C_DIS
LIN {X 0.191,Y -397.295,Z 752.599,A 0.000,B 0.000,C 90.000,E1 107.873} C_DIS
LIN {X 0.013,Y -414.584,Z 752.587,A 0.000,B 0.000,C 90.000,E1 105.662} C_DIS
LIN {X 0.042,Y -433.547,Z 752.575,A 0.000,B 0.000,C 90.000,E1 103.480} C_DIS
LIN {X 0.109,Y -453.620,Z 752.564,A 0.000,B 0.000,C 90.000,E1 101.422} C_DIS
LIN {X -0.056,Y -468.869,Z 752.556,A 0.000,B 0.000,C 90.000,E1 100.018} C_DIS
LIN {X -0.180,Y -470.779,Z 752.554,A 0.000,B 0.000,C 90.000,E1 99.792} C_DIS
LIN {X -0.225,Y -472.230,Z 752.553,A 0.000,B 0.000,C 90.000,E1 99.557} C_DIS
LIN {X -0.048,Y -474.210,Z 752.550,A 0.000,B 0.000,C 90.000,E1 99.029} C_DIS
LIN {X 0.064,Y -475.065,Z 752.547,A 0.000,B 0.000,C 90.000,E1 98.511} C_DIS
LIN {X 0.190,Y -474.944,Z 752.545,A 0.000,B 0.000,C 90.000,E1 97.992} C_DIS
LIN {X -0.148,Y -473.834,Z 752.542,A 0.000,B 0.000,C 90.000,E1 97.530} C_DIS
LIN {X 0.184,Y -472.858,Z 752.540,A 0.000,B 0.000,C 90.000,E1 97.239} C_DIS
LIN {X 0.043,Y -471.541,Z 752.539,A 0.000,B 0.000,C 90.000,E1 97.004} C_DIS
LIN {X -0.042,Y -452.211,Z 752.522,A 0.000,B 0.000,C 90.000,E1 93.955} C_DIS
LIN {X -0.211,Y -440.260,Z 752.510,A 0.000,B 0.000,C 90.000,E1 91.892} C_DIS
LIN {X 0.204,Y -432.691,Z 752.503,A 0.000,B 0.000,C 90.000,E1 90.516} C_DIS
LIN {X 0.192,Y -423.263,Z 752.494,A 0.000,B 0.000,C 90.000,E1 88.912} C_DIS
LIN {X 0.117,Y -412.192,Z 752.484,A 0.000,B 0.000,C 90.000,E1 87.020} C_DIS
LIN {X -0.132,Y -400.960,Z 752.473,A 0.000,B 0.000,C 90.000,E1 85.122} C_DIS
LIN {X -0.147,Y -388.133,Z 752.460,A 0.000,B 0.000,C 90.000,E1 82.875} C_DIS
LIN {X -0.036,Y -374.086,Z 752.446,A 0.000,B 0.000,C 90.000,E1 80.274} C_DIS
LIN {X -0.122,Y -360.652,Z 752.431,A 0.000,B 0.000,C 90.000,E1 77.645} C_DIS
LIN {X 0.075,Y -350.562,Z 752.420,A 0.000,B 0.000,C 90.000,E1 75.519} C_DIS
LIN {X 0.044,Y -339.263,Z 752.406,A 0.000,B 0.000,C 90.000,E1 73.087} C_DIS
LIN {X 0.004,Y -326.887,Z 752.391,A 0.000,B 0.000,C 90.000,E1 70.296} C_DIS
LIN {X 0.094,Y -313.925,Z 752.373,A 0.000,B 0.000,C 90.000,E1 67.102} C_DIS
LIN {X -0.131,Y -302.140,Z 752.355,A 0.000,B 0.000,C 90.000,E1 63.896} C_DIS
LIN {X 0.100,Y -290.519,Z 752.335,A 0.000,B 0.000,C 90.000,E1 60.205} C_DIS
LIN {X -0.030,Y -282.606,Z 752.320,A 0.000,B 0.000,C 90.000,E1 57.533} C_DIS
LIN {X 0.100,Y -274.995,Z 752.304,A 0.000,B 0.000,C 90.000,E1 54.769} C_DIS
LIN {X -0.035,Y -269.407,Z 752.293,A 0.000,B 0.000,C 90.000,E1 52.718} C_DIS
LIN {X 0.052,Y -263.813,Z 752.281,A 0.000,B 0.000,C 90.000,E1 50.598} C_DIS
LIN {X 0.066,Y -256.191,Z 752.265,A 0.000,B 0.000,C 90.000,E1 47.757} C_DIS
LIN {X -0.140,Y -250.483,Z 752.253,A 0.000,B 0.000,C 90.000,E1 45.648} C_DIS
LIN {X 0.059,Y -242.845,Z 752.237,A 0.000,B 0.000,C 90.000,E1 42.690} C_DIS
LIN {X 0.090,Y -235.210,Z 752.221,A 0.000,B 0.000,C 90.000,E1 39.725} C_DIS
LIN {X -0.099,Y -226.119,Z 752.200,A 0.000,B 0.000,C 90.000,E1 36.011} C_DIS
LIN {X 0.079,Y -217.753,Z 752.179,A 0.000,B 0.000,C 90.000,E1 32.133} C_DIS
LIN {X 0.050,Y -211.682,Z 752.161,A 0.000,B 0.000,C 90.000,E1 29.027} C_DIS
LIN {X -0.044,Y -206.446,Z 752.144,A 0.000,B 0.000,C 90.000,E1 25.899} C_DIS
LIN {X -0.005,Y -200.834,Z 752.122,A 0.000,B 0.000,C 90.000,E1 21.897} C_DIS
LIN {X -0.055,Y -196.316,Z 752.099,A 0.000,B 0.000,C 90.000,E1 17.873} C_DIS
LIN {X 0.074,Y -192.370,Z 752.072,A 0.000,B 0.000,C 90.000,E1 12.939} C_DIS
LIN {X 0.061,Y -189.617,Z 752.040,A 0.000,B 0.000,C 90.000,E1 7.182} C_DIS
LIN {X 0.005,Y -190.816,Z 751.965,A 0.000,B 0.000,C 90.000,E1 353.742} C_DIS
LIN {X -0.025,Y -193.880,Z 751.938,A 0.000,B 0.000,C 90.000,E1 348.814} C_DIS
LIN {X 0.070,Y -197.593,Z 751.915,A 0.000,B 0.000,C 90.000,E1 344.700} C_DIS
LIN {X -0.031,Y -202.227,Z 751.893,A 0.000,B 0.000,C 90.000,E1 340.678} C_DIS
LIN {X -0.019,Y -207.896,Z 751.870,A 0.000,B 0.000,C 90.000,E1 336.666} C_DIS
LIN {X 0.041,Y -214.393,Z 751.848,A 0.000,B 0.000,C 90.000,E1 332.692} C_DIS
LIN {X 0.043,Y -221.715,Z 751.827,A 0.000,B 0.000,C 90.000,E1 328.791} C_DIS
LIN {X -0.056,Y -229.597,Z 751.805,A 0.000,B 0.000,C 90.000,E1 324.975} C_DIS
LIN {X 0.056,Y -238.113,Z 751.784,A 0.000,B 0.000,C 90.000,E1 321.170} C_DIS
LIN {X 0.001,Y -247.361,Z 751.764,A 0.000,B 0.000,C 90.000,E1 317.472} C_DIS
LIN {X 0.027,Y -256.559,Z 751.746,A 0.000,B 0.000,C 90.000,E1 314.190} C_DIS
LIN {X 0.039,Y -267.648,Z 751.726,A 0.000,B 0.000,C 90.000,E1 310.620} C_DIS
LIN {X -0.087,Y -279.896,Z 751.706,A 0.000,B 0.000,C 90.000,E1 307.156} C_DIS
LIN {X -0.001,Y -290.533,Z 751.691,A 0.000,B 0.000,C 90.000,E1 304.405} C_DIS
LIN {X 0.034,Y -302.398,Z 751.676,A 0.000,B 0.000,C 90.000,E1 301.720} C_DIS
LIN {X -0.146,Y -319.131,Z 751.658,A 0.000,B 0.000,C 90.000,E1 298.487} C_DIS
LIN {X 0.000,Y -331.845,Z 751.646,A 0.000,B 0.000,C 90.000,E1 296.232} C_DIS
LIN {X -0.157,Y -345.277,Z 751.634,A 0.000,B 0.000,C 90.000,E1 294.079} C_DIS
LIN {X -0.134,Y -366.028,Z 751.617,A 0.000,B 0.000,C 90.000,E1 291.046} C_DIS
LIN {X 0.039,Y -384.174,Z 751.604,A 0.000,B 0.000,C 90.000,E1 288.671} C_DIS
LIN {X 0.065,Y -403.455,Z 751.591,A 0.000,B 0.000,C 90.000,E1 286.386} C_DIS
LIN {X 0.054,Y -415.367,Z 751.583,A 0.000,B 0.000,C 90.000,E1 285.009} C_DIS
LIN {X 0.177,Y -429.450,Z 751.574,A 0.000,B 0.000,C 90.000,E1 283.355} C_DIS
LIN {X -0.170,Y -440.816,Z 751.567,A 0.000,B 0.000,C 90.000,E1 282.063} C_DIS
LIN {X -0.167,Y -449.464,Z 751.561,A 0.000,B 0.000,C 90.000,E1 281.007} C_DIS
LIN {X 0.117,Y -459.715,Z 751.554,A 0.000,B 0.000,C 90.000,E1 279.670} C_DIS
LIN {X 0.037,Y -469.559,Z 751.547,A 0.000,B 0.000,C 90.000,E1 278.398} C_DIS
LIN {X -0.171,Y -476.852,Z 751.541,A 0.000,B 0.000,C 90.000,E1 277.409} C_DIS
LIN {X -0.235,Y -481.634,Z 751.537,A 0.000,B 0.000,C 90.000,E1 276.663} C_DIS
LIN {X -0.196,Y -485.610,Z 751.533,A 0.000,B 0.000,C 90.000,E1 275.910} C_DIS
LIN {X -0.176,Y -488.901,Z 751.529,A 0.000,B 0.000,C 90.000,E1 275.163} C_DIS
LIN {X 0.033,Y -490.614,Z 751.526,A 0.000,B 0.000,C 90.000,E1 274.645} C_DIS
LIN {X 0.211,Y -491.925,Z 751.523,A 0.000,B 0.000,C 90.000,E1 274.131} C_DIS
LIN {X -0.057,Y -492.815,Z 751.520,A 0.000,B 0.000,C 90.000,E1 273.669} C_DIS
LIN {X 0.145,Y -493.297,Z 751.518,A 0.000,B 0.000,C 90.000,E1 273.154} C_DIS
LIN {X -0.114,Y -493.384,Z 751.515,A 0.000,B 0.000,C 90.000,E1 272.694} C_DIS
LIN {X 0.099,Y -492.982,Z 751.512,A 0.000,B 0.000,C 90.000,E1 272.178} C_DIS
LIN {X -0.164,Y -492.202,Z 751.509,A 0.000,B 0.000,C 90.000,E1 271.718} C_DIS
LIN {X 0.047,Y -490.963,Z 751.507,A 0.000,B 0.000,C 90.000,E1 271.203} C_DIS
LIN {X -0.235,Y -489.195,Z 751.504,A 0.000,B 0.000,C 90.000,E1 270.745} C_DIS
LIN {X -0.034,Y -486.849,Z 751.501,A 0.000,B 0.000,C 90.000,E1 270.229} C_DIS
LIN {X 0.148,Y -483.873,Z 751.499,A 0.000,B 0.000,C 90.000,E1 269.714} C_DIS
LIN {X -0.166,Y -480.127,Z 751.496,A 0.000,B 0.000,C 90.000,E1 269.255} C_DIS
LIN {X -0.019,Y -475.509,Z 751.493,A 0.000,B 0.000,C 90.000,E1 268.740} C_DIS
LIN {X 0.131,Y -469.870,Z 751.490,A 0.000,B 0.000,C 90.000,E1 268.224} C_DIS
LIN {X 0.215,Y -466.954,Z 751.489,A 0.000,B 0.000,C 90.000,E1 267.993} C_DIS
LIN {X 0.156,Y -460.458,Z 751.487,A 0.000,B 0.000,C 90.000,E1 267.593} C_DIS
LIN {X 0.136,Y -453.626,Z 751.485,A 0.000,B 0.000,C 90.000,E1 267.249} C_DIS
LIN {X 0.169,Y -446.215,Z 751.483,A 0.000,B 0.000,C 90.000,E1 266.963} C_DIS
LIN {X -0.156,Y -438.390,Z 751.482,A 0.000,B 0.000,C 90.000,E1 266.788} C_DIS
LIN {X -0.059,Y -429.528,Z 751.481,A 0.000,B 0.000,C 90.000,E1 266.617} C_DIS
LIN {X -0.120,Y -422.908,Z 751.481,A 0.000,B 0.000,C 90.000,E1 266.560} C_DIS
LIN {X 0.160,Y -418.579,Z 751.481,A 0.000,B 0.000,C 90.000,E1 266.502} C_DIS
LIN {X 0.040,Y -180.950,Z 751.481,A 0.000,B 0.000,C 90.000,E1 266.502} C_DIS
LIN {X 0.005,Y -180.798,Z 751.471,A 0.000,B 0.000,C 90.000,E1 264.780} C_DIS
LIN {X 0.079,Y -178.898,Z 751.443,A 0.000,B 0.000,C 90.000,E1 259.690} C_DIS
LIN {X -0.016,Y -175.941,Z 751.415,A 0.000,B 0.000,C 90.000,E1 254.629} C_DIS
LIN {X -0.070,Y -175.396,Z 751.410,A 0.000,B 0.000,C 90.000,E1 253.795} C_DIS
LIN {X -0.065,Y -172.165,Z 751.386,A 0.000,B 0.000,C 90.000,E1 249.518} C_DIS
LIN {X -0.026,Y -171.634,Z 751.381,A 0.000,B 0.000,C 90.000,E1 248.646} C_DIS
LIN {X -0.031,Y -167.857,Z 751.357,A 0.000,B 0.000,C 90.000,E1 244.332} C_DIS
LIN {X -0.088,Y -166.588,Z 751.348,A 0.000,B 0.000,C 90.000,E1 242.615} C_DIS
LIN {X 0.046,Y -162.578,Z 751.323,A 0.000,B 0.000,C 90.000,E1 238.201} C_DIS
LIN {X 0.105,Y -161.261,Z 751.314,A 0.000,B 0.000,C 90.000,E1 236.421} C_DIS
LIN {X 0.015,Y -157.263,Z 751.289,A 0.000,B 0.000,C 90.000,E1 232.029} C_DIS
LIN {X -0.058,Y -155.983,Z 751.279,A 0.000,B 0.000,C 90.000,E1 230.275} C_DIS
LIN {X -0.098,Y -152.239,Z 751.254,A 0.000,B 0.000,C 90.000,E1 225.810} C_DIS
LIN {X 0.028,Y -150.480,Z 751.239,A 0.000,B 0.000,C 90.000,E1 223.056} C_DIS
LIN {X -0.044,Y -147.205,Z 751.214,A 0.000,B 0.000,C 90.000,E1 218.543} C_DIS
LIN {X -0.073,Y -145.225,Z 751.194,A 0.000,B 0.000,C 90.000,E1 214.898} C_DIS
LIN {X 0.038,Y -142.352,Z 751.163,A 0.000,B 0.000,C 90.000,E1 209.333} C_DIS
LIN {X -0.035,Y -141.740,Z 751.153,A 0.000,B 0.000,C 90.000,E1 207.513} C_DIS
